short summary
=================
Returns the interface :ref:`ISimpleDateAndTimeAssertions`
with assert statements for date and time types with 32 bit length

.. <legal notes>

legal notes
=================
| SPDX-FileCopyrightText: © 2022 ekvip automation GmbH <info@ekvip.de>
| SPDX-License-Identifier: Apache-2.0
| For details check: Apache-2.0_

.. _Apache-2.0: https://www.apache.org/licenses/LICENSE-2.0

.. </legal notes>

methods
==================

*)

PROPERTY simple :ISimpleDateAndTimeAssertions
GET
simple := THIS^.assertionsFor32BitTypes;
END_GET
END_PROPERTY

END_FUNCTION_BLOCK

// ---- Assertor/Assertions/DateAndTimeAssertions/32Bit/classes/SimpleDateAndTimeAssertions.TcPOU
(*

short summary
=================
| This class provides assert statements for date and time types with 32 bit length
| It implements the interface :ref:`ISimpleDateAndTimeAssertions`
| For date and time (``DT``) use :ref:`SimpleDateAndTimeAssertions.dateAndTime`
| For date (``DATE``) use  :ref:`SimpleDateAndTimeAssertions.dateOnly`
| For time of day (``TOD``) use  :ref:`SimpleDateAndTimeAssertions.timeOfDay`

.. <legal notes>

legal notes
=================
| SPDX-FileCopyrightText: © 2022 ekvip automation GmbH <info@ekvip.de>
| SPDX-License-Identifier: Apache-2.0
| For details check: Apache-2.0_

.. _Apache-2.0: https://www.apache.org/licenses/LICENSE-2.0

.. </legal notes>

methods and properties
=======================

*)

{attribute 'reflection'}
FUNCTION_BLOCK INTERNAL SimpleDateAndTimeAssertions 
EXTENDS CNM_AbstractObject.Object
IMPLEMENTS ISimpleDateAndTimeAssertions, IAssertCallBacksetter
VAR
	(* class to handle date assertions *)
	dateAssertions		:DateAssertions32Bit();
	(* class to handle date and time assertions *)
	dateTimeAssertions	:DateTimeAssertions32Bit();
	(* class to handle time of day assertions *)
	timeOfDayAssertions	:TimeOfDayAssertions32Bit();
END_VAR

(*

short summary
=================
This abstract property returns the class name of the concrete object, 
It's for debugging purpose

.. <legal notes>

legal notes
=================
| SPDX-FileCopyrightText: © 2022 ekvip automation GmbH <info@ekvip.de>
| SPDX-License-Identifier: Apache-2.0
| For details check: Apache-2.0_

.. _Apache-2.0: https://www.apache.org/licenses/LICENSE-2.0

.. </legal notes>

*)

PROPERTY className :CNM_AbstractObject.ClassName
GET
className := 'CNM_AssertionInterfaceLib.SimplyDateAndTimeAssertions';
END_GET
END_PROPERTY

(*

short summary
=================
Returns the interface :ref:`I32BitDtAssertions`
with assert statements for 32 bit date and time ``DT``

.. <legal notes>

legal notes
=================
| SPDX-FileCopyrightText: © 2022 ekvip automation GmbH <info@ekvip.de>
| SPDX-License-Identifier: Apache-2.0
| For details check: Apache-2.0_

.. _Apache-2.0: https://www.apache.org/licenses/LICENSE-2.0

.. </legal notes>

*)

PROPERTY dateAndTime :I32BitDtAssertions
GET
dateAndTime := THIS^.dateTimeAssertions;
END_GET
END_PROPERTY

(*

short summary
=================
Returns the interface :ref:`I32BitDateAssertions`
with assert statements for 32 bit date ``DATE``

.. <legal notes>

legal notes
=================
| SPDX-FileCopyrightText: © 2022 ekvip automation GmbH <info@ekvip.de>
| SPDX-License-Identifier: Apache-2.0
| For details check: Apache-2.0_

.. _Apache-2.0: https://www.apache.org/licenses/LICENSE-2.0

.. </legal notes>

*)

PROPERTY dateOnly : I32BitDateAssertions
GET
dateOnly := THIS^.dateAssertions;
END_GET
END_PROPERTY

(*

short summary
=================
This methods is the setter for the callback class if an assertion was false

.. <legal notes>

legal notes
=================
| SPDX-FileCopyrightText: © 2022 ekvip automation GmbH <info@ekvip.de>
| SPDX-License-Identifier: Apache-2.0
| For details check: Apache-2.0_

.. _Apache-2.0: https://www.apache.org/licenses/LICENSE-2.0

.. </legal notes>

parameters
=================

*)

METHOD setCallBack
VAR_INPUT
	(* the class that must be informed if an assertion is false *)
	callBack	:IAssertCallback;  
END_VAR
THIS^.dateAssertions.setCallBack(callBack);
THIS^.dateTimeAssertions.setCallBack(callBack);
THIS^.timeOfDayAssertions.setCallBack(callBack);
END_METHOD

(*

short summary
=================
Returns the interface :ref:`I32BitDateAssertions`
with assert statements for 32 bit time of day ``TOD``

.. <legal notes>

legal notes
=================
| SPDX-FileCopyrightText: © 2022 ekvip automation GmbH <info@ekvip.de>
| SPDX-License-Identifier: Apache-2.0
| For details check: Apache-2.0_

.. _Apache-2.0: https://www.apache.org/licenses/LICENSE-2.0

.. </legal notes>

*)

PROPERTY timeOfDay :I32BitTodAssertions
GET
timeOfDay := THIS^.timeOfDayAssertions;
END_GET
END_PROPERTY

END_FUNCTION_BLOCK

// ---- Assertor/Assertions/DateAndTimeAssertions/32Bit/Date/classes/DateAssertions32Bit.TcPOU
(*

short summary
=================
This class provides assert statements for 32 bit ``DATE``.
It implements :ref:`I32BitDateAssertions`

.. <legal notes>

legal notes
=================
| SPDX-FileCopyrightText: © 2022 ekvip automation GmbH <info@ekvip.de>
| SPDX-License-Identifier: Apache-2.0
| For details check: Apache-2.0_

.. _Apache-2.0: https://www.apache.org/licenses/LICENSE-2.0

.. </legal notes>

methods and properties
=======================

*)

{attribute 'reflection'}
FUNCTION_BLOCK INTERNAL DateAssertions32Bit EXTENDS AbstactAssertion IMPLEMENTS I32BitDateAssertions
VAR
END_VAR

(*

short summary
=================
This abstract property returns the class name of the concrete object, 
It's for debugging purpose

.. <legal notes>

legal notes
=================
| SPDX-FileCopyrightText: © 2022 ekvip automation GmbH <info@ekvip.de>
| SPDX-License-Identifier: Apache-2.0
| For details check: Apache-2.0_

.. _Apache-2.0: https://www.apache.org/licenses/LICENSE-2.0

.. </legal notes>

*)

PROPERTY className :CNM_AbstractObject.ClassName
GET
className := 'CNM_AssertionInterfaceLib.DateAssertions32Bit';
END_GET
END_PROPERTY

(*

short summary
=================
This assertion method checks if the current value is equal to the expected value

.. <legal notes>

legal notes
=================
| SPDX-FileCopyrightText: © 2022 ekvip automation GmbH <info@ekvip.de>
| SPDX-License-Identifier: Apache-2.0
| For details check: Apache-2.0_

.. _Apache-2.0: https://www.apache.org/licenses/LICENSE-2.0

.. </legal notes>

parameters
=================

*)

METHOD valueIsEqualTo
VAR_INPUT
	(* current value to check *)
	currentValue	:DATE;
	(* expected value to compare *)
	expectedValue	:DATE;
	(* message if the assertion is false *)
	message			:AssertMessage;
END_VAR
IF (currentValue <> expectedValue) THEN
	THIS^.assertionWasWrong(message, THIS^.getDebugInfo('valueIsEqualTo'));
END_IF
END_METHOD

(*

short summary
=================
This assertion method checks if the current value is greater than the less value

.. <legal notes>

legal notes
=================
| SPDX-FileCopyrightText: © 2022 ekvip automation GmbH <info@ekvip.de>
| SPDX-License-Identifier: Apache-2.0
| For details check: Apache-2.0_

.. _Apache-2.0: https://www.apache.org/licenses/LICENSE-2.0

.. </legal notes>

parameters
=================

*)

METHOD valueIsGreaterThan
VAR_INPUT
	(* current value to check *)
	currentValue	:DATE;
	(* less than lower limit *)
	lessValue		:DATE;
	(* message if the assertion is false *)
	message			:AssertMessage;
END_VAR
IF (currentValue <= lessValue) THEN
	THIS^.assertionWasWrong(message, THIS^.getDebugInfo('valueIsGreaterThan'));
END_IF
END_METHOD

(*

short summary
=================
This assertion method checks if the current value is inside a limit

.. attention:: 
	limits are included: ``valueIsInRangeOf(date#1970-01-01, date#1970-01-01, date#1970-01-01)``
	is a true assertion

.. <legal notes>

legal notes
=================
| SPDX-FileCopyrightText: © 2022 ekvip automation GmbH <info@ekvip.de>
| SPDX-License-Identifier: Apache-2.0
| For details check: Apache-2.0_

.. _Apache-2.0: https://www.apache.org/licenses/LICENSE-2.0

.. </legal notes>

parameters
=================

*)

METHOD valueIsInRangeOf
VAR_INPUT
	(* lower limit for the current value *)
	lowerLimit		:DATE;
	(* current value to check *)
	currentValue	:DATE;
	(* upper limit for the current value *)
	upperLimit		:DATE;
	(* message if the assertion is false *)
	message			:AssertMessage;
END_VAR
IF (
	(currentValue < lowerLimit)
	OR (currentValue > upperLimit)
) THEN
	THIS^.assertionWasWrong(message, THIS^.getDebugInfo('valueIsInRangeOf'));
END_IF
END_METHOD

(*

short summary
=================
This assertion method checks if the current value is less than the greater value

.. <legal notes>

legal notes
=================
| SPDX-FileCopyrightText: © 2022 ekvip automation GmbH <info@ekvip.de>
| SPDX-License-Identifier: Apache-2.0
| For details check: Apache-2.0_

.. _Apache-2.0: https://www.apache.org/licenses/LICENSE-2.0

.. </legal notes>

parameters
=================

*)

METHOD valueIsLessThan
VAR_INPUT
	(* current value to check *)
	currentValue	:DATE;
	(* greater than upper limit *)
	greaterValue	:DATE;
	(* message if the assertion is false *)
	message			:AssertMessage;
END_VAR
IF (currentValue >= greaterValue) THEN
	THIS^.assertionWasWrong(message, THIS^.getDebugInfo('valueIsLessThan'));
END_IF
END_METHOD

(*

short summary
=================
This assertion method checks if the current value is less than or equal to the maximum value

.. <legal notes>

legal notes
=================
| SPDX-FileCopyrightText: © 2022 ekvip automation GmbH <info@ekvip.de>
| SPDX-License-Identifier: Apache-2.0
| For details check: Apache-2.0_

.. _Apache-2.0: https://www.apache.org/licenses/LICENSE-2.0

.. </legal notes>

parameters
=================

*)

METHOD valueIsMax
VAR_INPUT
	(* current value to check *)
	currentValue	:DATE;
	(* upper limit for the current value *)
	maximumValue	:DATE;
	(* message if the assertion is false *)
	message			:AssertMessage;
END_VAR
IF (currentValue > maximumValue) THEN
	THIS^.assertionWasWrong(message, THIS^.getDebugInfo('valueIsMax'));
END_IF
END_METHOD

(*

short summary
=================
This assertion method checks if the current value is greater than or equal to the minimum value

.. <legal notes>

legal notes
=================
| SPDX-FileCopyrightText: © 2022 ekvip automation GmbH <info@ekvip.de>
| SPDX-License-Identifier: Apache-2.0
| For details check: Apache-2.0_

.. _Apache-2.0: https://www.apache.org/licenses/LICENSE-2.0

.. </legal notes>

parameters
=================

*)

METHOD valueIsMin
VAR_INPUT
	(* current value to check *)
	currentValue	:DATE;
	(* lower limit for the current value *)
	minimumValue	:DATE;
	(* message if the assertion is false *)
	message			:AssertMessage;
END_VAR
IF (currentValue < minimumValue) THEN
	THIS^.assertionWasWrong(message, THIS^.getDebugInfo('valueIsMin'));
END_IF
END_METHOD

(*

short summary
=================
This assertion method checks if the current value is not equal to the unexpected value

.. <legal notes>

legal notes
=================
| SPDX-FileCopyrightText: © 2022 ekvip automation GmbH <info@ekvip.de>
| SPDX-License-Identifier: Apache-2.0
| For details check: Apache-2.0_

.. _Apache-2.0: https://www.apache.org/licenses/LICENSE-2.0

.. </legal notes>

parameters
=================

*)

METHOD valueIsNotEqualTo
VAR_INPUT
	(* current value to check *)
	currentValue	:DATE;
	(* unexpected value to compare *)
	unexpectedValue	:DATE;
	(* message if the assertion is false *)
	message			:AssertMessage;
END_VAR
IF (currentValue = unexpectedValue) THEN
	THIS^.assertionWasWrong(message, THIS^.getDebugInfo('valueIsNotEqualTo'));
END_IF
END_METHOD

END_FUNCTION_BLOCK

// ---- Assertor/Assertions/DateAndTimeAssertions/32Bit/DT/classes/DateTimeAssertions32Bit.TcPOU
(*

short summary
=================
This class provides assert statements for 32 bit date and time ``DT``.
It implements the interface :ref:`I32BitDtAssertions` 

.. <legal notes>

legal notes
=================
| SPDX-FileCopyrightText: © 2022 ekvip automation GmbH <info@ekvip.de>
| SPDX-License-Identifier: Apache-2.0
| For details check: Apache-2.0_

.. _Apache-2.0: https://www.apache.org/licenses/LICENSE-2.0

.. </legal notes>

methods and properties
=======================

*)

{attribute 'reflection'}
FUNCTION_BLOCK INTERNAL DateTimeAssertions32Bit EXTENDS AbstactAssertion IMPLEMENTS I32BitDtAssertions
VAR
END_VAR

(*

short summary
=================
This abstract property returns the class name of the concrete object, 
It's for debugging purpose

.. <legal notes>

legal notes
=================
| SPDX-FileCopyrightText: © 2022 ekvip automation GmbH <info@ekvip.de>
| SPDX-License-Identifier: Apache-2.0
| For details check: Apache-2.0_

.. _Apache-2.0: https://www.apache.org/licenses/LICENSE-2.0

.. </legal notes>

*)

PROPERTY className :CNM_AbstractObject.ClassName
GET
className := 'CNM_AssertionInterfaceLib.DateTimeAssertions32Bit';
END_GET
END_PROPERTY

(*

short summary
=================
This assertion method checks if the current value is equal to the expected value

.. <legal notes>

legal notes
=================
| SPDX-FileCopyrightText: © 2022 ekvip automation GmbH <info@ekvip.de>
| SPDX-License-Identifier: Apache-2.0
| For details check: Apache-2.0_

.. _Apache-2.0: https://www.apache.org/licenses/LICENSE-2.0

.. </legal notes>

parameters
=================

*)

METHOD valueIsEqualTo
VAR_INPUT
	(* current value to check *)
	currentValue	:DT;
	(* expected value to compare *)
	expectedValue	:DT;
	(* message if the assertion is false *)
	message			:AssertMessage;
END_VAR
IF (currentValue <> expectedValue) THEN
	THIS^.assertionWasWrong(message, THIS^.getDebugInfo('valueIsEqualTo'));
END_IF
END_METHOD

(*

short summary
=================
This assertion method checks if the current value is greater than the less value

.. <legal notes>

legal notes
=================
| SPDX-FileCopyrightText: © 2022 ekvip automation GmbH <info@ekvip.de>
| SPDX-License-Identifier: Apache-2.0
| For details check: Apache-2.0_

.. _Apache-2.0: https://www.apache.org/licenses/LICENSE-2.0

.. </legal notes>

parameters
=================

*)

METHOD valueIsGreaterThan
VAR_INPUT
	(* current value to check *)
	currentValue	:DT;
	(* less than lower limit *)
	lessValue		:DT;
	(* message if the assertion is false *)
	message			:AssertMessage;
END_VAR
IF (currentValue <= lessValue) THEN
	THIS^.assertionWasWrong(message, THIS^.getDebugInfo('valueIsGreaterThan'));
END_IF
END_METHOD

(*

short summary
=================
This assertion method checks if the current value is inside a limit

.. attention:: 
	limits are included: ``valueIsInRangeOf(dt#1970-01-01-0:0:0, dt#1970-01-01-0:0:0, dt#1970-01-01-0:0:0)``
	is a true assertion

.. <legal notes>

legal notes
=================
| SPDX-FileCopyrightText: © 2022 ekvip automation GmbH <info@ekvip.de>
| SPDX-License-Identifier: Apache-2.0
| For details check: Apache-2.0_

.. _Apache-2.0: https://www.apache.org/licenses/LICENSE-2.0

.. </legal notes>

parameters
=================

*)

METHOD valueIsInRangeOf
VAR_INPUT
	(* lower limit for the current value *)
	lowerLimit		:DT;
	(* current value to check *)
	currentValue	:DT;
	(* upper limit for the current value *)
	upperLimit		:DT;
	(* message if the assertion is false *)
	message			:AssertMessage;
END_VAR
IF (
	(currentValue < lowerLimit)
	OR (currentValue > upperLimit)
) THEN
	THIS^.assertionWasWrong(message, THIS^.getDebugInfo('valueIsInRangeOf'));
END_IF
END_METHOD

(*

short summary
=================
This assertion method checks if the current value is less than the greater value

.. <legal notes>

legal notes
=================
| SPDX-FileCopyrightText: © 2022 ekvip automation GmbH <info@ekvip.de>
| SPDX-License-Identifier: Apache-2.0
| For details check: Apache-2.0_

.. _Apache-2.0: https://www.apache.org/licenses/LICENSE-2.0

.. </legal notes>

parameters
=================

*)

METHOD valueIsLessThan
VAR_INPUT
	(* current value to check *)
	currentValue	:DT;
	(* greater than upper limit *)
	greaterValue	:DT;
	(* message if the assertion is false *)
	message			:AssertMessage;
END_VAR
IF (currentValue >= greaterValue) THEN
	THIS^.assertionWasWrong(message, THIS^.getDebugInfo('valueIsLessThan'));
END_IF
END_METHOD

(*

short summary
=================
This assertion method checks if the current value is less than or equal to the maximum value

.. <legal notes>

legal notes
=================
| SPDX-FileCopyrightText: © 2022 ekvip automation GmbH <info@ekvip.de>
| SPDX-License-Identifier: Apache-2.0
| For details check: Apache-2.0_

.. _Apache-2.0: https://www.apache.org/licenses/LICENSE-2.0

.. </legal notes>

parameters
=================

*)

METHOD valueIsMax
VAR_INPUT
	(* current value to check *)
	currentValue	:DT;
	(* upper limit for the current value *)
	maximumValue	:DT;
	(* message if the assertion is false *)
	message			:AssertMessage;
END_VAR
IF (currentValue > maximumValue) THEN
	THIS^.assertionWasWrong(message, THIS^.getDebugInfo('valueIsMax'));
END_IF
END_METHOD

(*

short summary
=================
This assertion method checks if the current value is greater than or equal to the minimum value

.. <legal notes>

legal notes
=================
| SPDX-FileCopyrightText: © 2022 ekvip automation GmbH <info@ekvip.de>
| SPDX-License-Identifier: Apache-2.0
| For details check: Apache-2.0_

.. _Apache-2.0: https://www.apache.org/licenses/LICENSE-2.0

.. </legal notes>

parameters
=================

*)

METHOD valueIsMin
VAR_INPUT
	(* current value to check *)
	currentValue	:DT;
	(* lower limit for the current value *)
	minimumValue	:DT;
	(* message if the assertion is false *)
	message			:AssertMessage;
END_VAR
IF (currentValue < minimumValue) THEN
	THIS^.assertionWasWrong(message, THIS^.getDebugInfo('valueIsMin'));
END_IF
END_METHOD

(*

short summary
=================
This assertion method checks if the current value is not equal to the unexpected value

.. <legal notes>

legal notes
=================
| SPDX-FileCopyrightText: © 2022 ekvip automation GmbH <info@ekvip.de>
| SPDX-License-Identifier: Apache-2.0
| For details check: Apache-2.0_

.. _Apache-2.0: https://www.apache.org/licenses/LICENSE-2.0

.. </legal notes>

parameters
=================

*)

METHOD valueIsNotEqualTo
VAR_INPUT
	(* current value to check *)
	currentValue	:DT;
	(* unexpected value to compare *)
	unexpectedValue	:DT;
	(* message if the assertion is false *)
	message			:AssertMessage;
END_VAR
IF (currentValue = unexpectedValue) THEN
	THIS^.assertionWasWrong(message, THIS^.getDebugInfo('valueIsNotEqualTo'));
END_IF
END_METHOD

END_FUNCTION_BLOCK

// ---- Assertor/Assertions/DateAndTimeAssertions/32Bit/TOD/classes/TimeOfDayAssertions32Bit.TcPOU
(*

short summary
=================
This class provides assert statements for 32 bit time of day ``TOD``.
It implements the interface :ref:`I32BitTodAssertions`

.. <legal notes>

legal notes
=================
| SPDX-FileCopyrightText: © 2022 ekvip automation GmbH <info@ekvip.de>
| SPDX-License-Identifier: Apache-2.0
| For details check: Apache-2.0_

.. _Apache-2.0: https://www.apache.org/licenses/LICENSE-2.0

.. </legal notes>

methods
==================

*)

{attribute 'reflection'}
FUNCTION_BLOCK INTERNAL TimeOfDayAssertions32Bit EXTENDS AbstactAssertion IMPLEMENTS I32BitTodAssertions
VAR
END_VAR

(*

short summary
=================
This abstract property returns the class name of the concrete object, 
It's for debugging purpose

.. <legal notes>

legal notes
=================
| SPDX-FileCopyrightText: © 2022 ekvip automation GmbH <info@ekvip.de>
| SPDX-License-Identifier: Apache-2.0
| For details check: Apache-2.0_

.. _Apache-2.0: https://www.apache.org/licenses/LICENSE-2.0

.. </legal notes>

*)

PROPERTY className :CNM_AbstractObject.ClassName
GET
className := 'CNM_AssertionInterfaceLib.TimeOfDayAssertions32Bit';
END_GET
END_PROPERTY

(*

short summary
=================
This assertion method checks if the current value is equal to the expected value

.. <legal notes>

legal notes
=================
| SPDX-FileCopyrightText: © 2022 ekvip automation GmbH <info@ekvip.de>
| SPDX-License-Identifier: Apache-2.0
| For details check: Apache-2.0_

.. _Apache-2.0: https://www.apache.org/licenses/LICENSE-2.0

.. </legal notes>

parameters
=================

*)

METHOD valueIsEqualTo
VAR_INPUT
	(* current value to check *)
	currentValue	:TOD;
	(* expected value to compare *)
	expectedValue	:TOD;
	(* message if the assertion is false *)
	message			:AssertMessage;
END_VAR
IF (currentValue <> expectedValue) THEN
	THIS^.assertionWasWrong(message, THIS^.getDebugInfo('valueIsEqualTo'));
END_IF
END_METHOD

(*

short summary
=================
This assertion method checks if the current value is greater than the less value

.. <legal notes>

legal notes
=================
| SPDX-FileCopyrightText: © 2022 ekvip automation GmbH <info@ekvip.de>
| SPDX-License-Identifier: Apache-2.0
| For details check: Apache-2.0_

.. _Apache-2.0: https://www.apache.org/licenses/LICENSE-2.0

.. </legal notes>

parameters
=================

*)

METHOD valueIsGreaterThan
VAR_INPUT
	(* current value to check *)
	currentValue	:TOD;
	(* less than lower limit *)
	lessValue		:TOD;
	(* message if the assertion is false *)
	message			:AssertMessage;
END_VAR
IF (currentValue <= lessValue) THEN
	THIS^.assertionWasWrong(message, THIS^.getDebugInfo('valueIsGreaterThan'));
END_IF
END_METHOD

(*

short summary
=================
This assertion method checks if the current value is inside a limit

.. attention:: 
	limits are included: ``valueIsInRangeOf(tod#3:0:0, tod#3:0:0, tod#3:0:0)`` is a true assertion

.. <legal notes>

legal notes
=================
| SPDX-FileCopyrightText: © 2022 ekvip automation GmbH <info@ekvip.de>
| SPDX-License-Identifier: Apache-2.0
| For details check: Apache-2.0_

.. _Apache-2.0: https://www.apache.org/licenses/LICENSE-2.0

.. </legal notes>

parameters
=================

*)

METHOD valueIsInRangeOf
VAR_INPUT
	(* lower limit for the current value *)
	lowerLimit		:TOD;
	(* current value to check *)
	currentValue	:TOD;
	(* upper limit for the current value *)
	upperLimit		:TOD;
	(* message if the assertion is false *)
	message			:AssertMessage;
END_VAR
IF (
	(currentValue < lowerLimit)
	OR (currentValue > upperLimit)
) THEN
	THIS^.assertionWasWrong(message, THIS^.getDebugInfo('valueIsInRangeOf'));
END_IF
END_METHOD

(*

short summary
=================
This assertion method checks if the current value is less than the greater value

.. <legal notes>

legal notes
=================
| SPDX-FileCopyrightText: © 2022 ekvip automation GmbH <info@ekvip.de>
| SPDX-License-Identifier: Apache-2.0
| For details check: Apache-2.0_

.. _Apache-2.0: https://www.apache.org/licenses/LICENSE-2.0

.. </legal notes>

parameters
=================

*)

METHOD valueIsLessThan
VAR_INPUT
	(* current value to check *)
	currentValue	:TOD;
	(* greater than upper limit *)
	greaterValue	:TOD;
	(* message if the assertion is false *)
	message			:AssertMessage;
END_VAR
IF (currentValue >= greaterValue) THEN
	THIS^.assertionWasWrong(message, THIS^.getDebugInfo('valueIsLessThan'));
END_IF
END_METHOD

(*

short summary
=================
This assertion method checks if the current value is less than or equal to the maximum value

.. <legal notes>

legal notes
=================
| SPDX-FileCopyrightText: © 2022 ekvip automation GmbH <info@ekvip.de>
| SPDX-License-Identifier: Apache-2.0
| For details check: Apache-2.0_

.. _Apache-2.0: https://www.apache.org/licenses/LICENSE-2.0

.. </legal notes>

parameters
=================

*)

METHOD valueIsMax
VAR_INPUT
	(* current value to check *)
	currentValue	:TOD;
	(* upper limit for the current value *)
	maximumValue	:TOD;
	(* message if the assertion is false *)
	message			:AssertMessage;
END_VAR
IF (currentValue > maximumValue) THEN
	THIS^.assertionWasWrong(message, THIS^.getDebugInfo('valueIsMax'));
END_IF
END_METHOD

(*

short summary
=================
This assertion method checks if the current value is greater than or equal to the minimum value

.. <legal notes>

legal notes
=================
| SPDX-FileCopyrightText: © 2022 ekvip automation GmbH <info@ekvip.de>
| SPDX-License-Identifier: Apache-2.0
| For details check: Apache-2.0_

.. _Apache-2.0: https://www.apache.org/licenses/LICENSE-2.0

.. </legal notes>

parameters
=================

*)

METHOD valueIsMin
VAR_INPUT
	(* current value to check *)
	currentValue	:TOD;
	(* lower limit for the current value *)
	minimumValue	:TOD;
	(* message if the assertion is false *)
	message			:AssertMessage;
END_VAR
IF (currentValue < minimumValue) THEN
	THIS^.assertionWasWrong(message, THIS^.getDebugInfo('valueIsMin'));
END_IF
END_METHOD

(*

short summary
=================
This assertion method checks if the current value is not equal to the unexpected value

.. <legal notes>

legal notes
=================
| SPDX-FileCopyrightText: © 2022 ekvip automation GmbH <info@ekvip.de>
| SPDX-License-Identifier: Apache-2.0
| For details check: Apache-2.0_

.. _Apache-2.0: https://www.apache.org/licenses/LICENSE-2.0

.. </legal notes>

parameters
=================

*)

METHOD valueIsNotEqualTo
VAR_INPUT
	(* current value to check *)
	currentValue	:TOD;
	(* unexpected value to compare *)
	unexpectedValue	:TOD;
	(* message if the assertion is false *)
	message			:AssertMessage;
END_VAR
IF (currentValue = unexpectedValue) THEN
	THIS^.assertionWasWrong(message, THIS^.getDebugInfo('valueIsNotEqualTo'));
END_IF
END_METHOD

END_FUNCTION_BLOCK

// ---- Assertor/Assertions/DateAndTimeAssertions/64Bit/classes/LongDateAndTimeAssertions.TcPOU
(*

short summary
=================
| This class provides assert statements for date and time types with 32 bit length
| It implements the interface :ref:`ISimpleDateAndTimeAssertions`
| For date and time (``DT``) use :ref:`SimpleDateAndTimeAssertions.dateAndTime`
| For date (``DATE``) use  :ref:`SimpleDateAndTimeAssertions.dateOnly`
| For time of day (``TOD``) use  :ref:`SimpleDateAndTimeAssertions.timeOfDay`

.. <legal notes>

legal notes
=================
| SPDX-FileCopyrightText: © 2022 ekvip automation GmbH <info@ekvip.de>
| SPDX-License-Identifier: Apache-2.0
| For details check: Apache-2.0_

.. _Apache-2.0: https://www.apache.org/licenses/LICENSE-2.0

.. </legal notes>

methods and properties
=======================

*)

{attribute 'reflection'}
FUNCTION_BLOCK INTERNAL LongDateAndTimeAssertions 
EXTENDS CNM_AbstractObject.Object
IMPLEMENTS ILongDateAndTimeAssertions, IAssertCallBacksetter
VAR
	(* class to handle date assertions *)
	dateAssertions		:DateAssertions64Bit();
	(* class to handle date and time assertions *)
	dateTimeAssertions	:DateTimeAssertions64Bit();
	(* class to handle time of day assertions *)
	timeOfDayAssertions	:TimeOfDayAssertions64Bit();
END_VAR

(*

short summary
=================
This abstract property returns the class name of the concrete object, 
It's for debugging purpose

.. <legal notes>

legal notes
=================
| SPDX-FileCopyrightText: © 2022 ekvip automation GmbH <info@ekvip.de>
| SPDX-License-Identifier: Apache-2.0
| For details check: Apache-2.0_

.. _Apache-2.0: https://www.apache.org/licenses/LICENSE-2.0

.. </legal notes>

*)

PROPERTY className :CNM_AbstractObject.ClassName
GET
className := 'CNM_AssertionInterfaceLib.SimplyDateAndTimeAssertions';
END_GET
END_PROPERTY

(*

short summary
=================
Returns the interface :ref:`I32BitDtAssertions`
with assert statements for 32 bit date and time ``DT``

.. <legal notes>

legal notes
=================
| SPDX-FileCopyrightText: © 2022 ekvip automation GmbH <info@ekvip.de>
| SPDX-License-Identifier: Apache-2.0
| For details check: Apache-2.0_

.. _Apache-2.0: https://www.apache.org/licenses/LICENSE-2.0

.. </legal notes>

*)

PROPERTY dateAndTime :I64BitDtAssertions
GET
dateAndTime := THIS^.dateTimeAssertions;
END_GET
END_PROPERTY

(*

short summary
=================
Returns the interface :ref:`I32BitDateAssertions`
with assert statements for 32 bit date ``DATE``

.. <legal notes>

legal notes
=================
| SPDX-FileCopyrightText: © 2022 ekvip automation GmbH <info@ekvip.de>
| SPDX-License-Identifier: Apache-2.0
| For details check: Apache-2.0_

.. _Apache-2.0: https://www.apache.org/licenses/LICENSE-2.0

.. </legal notes>

*)

PROPERTY dateOnly : I64BitDateAssertions
GET
dateOnly := THIS^.dateAssertions;
END_GET
END_PROPERTY

(*

short summary
=================
This methods is the setter for the callback class if an assertion was false

.. <legal notes>

legal notes
=================
| SPDX-FileCopyrightText: © 2022 ekvip automation GmbH <info@ekvip.de>
| SPDX-License-Identifier: Apache-2.0
| For details check: Apache-2.0_

.. _Apache-2.0: https://www.apache.org/licenses/LICENSE-2.0

.. </legal notes>

parameters
=================

*)

METHOD setCallBack
VAR_INPUT
	(* the class that must be informed if an assertion is false *)
	callBack	:IAssertCallback;  
END_VAR
THIS^.dateAssertions.setCallBack(callBack);
THIS^.dateTimeAssertions.setCallBack(callBack);
THIS^.timeOfDayAssertions.setCallBack(callBack);
END_METHOD

(*

short summary
=================
Returns the interface :ref:`I32BitDateAssertions`
with assert statements for 32 bit time of day ``TOD``

.. <legal notes>

legal notes
=================
| SPDX-FileCopyrightText: © 2022 ekvip automation GmbH <info@ekvip.de>
| SPDX-License-Identifier: Apache-2.0
| For details check: Apache-2.0_

.. _Apache-2.0: https://www.apache.org/licenses/LICENSE-2.0

.. </legal notes>

*)

PROPERTY timeOfDay :I64BitTodAssertions
GET
timeOfDay := THIS^.timeOfDayAssertions;
END_GET
END_PROPERTY

END_FUNCTION_BLOCK

// ---- Assertor/Assertions/DateAndTimeAssertions/64Bit/LDate/classes/DateAssertions64Bit.TcPOU
(*

short summary
=================
This class provides assert statements for 64 bit ``LDATE``.
It implements :ref:`I64BitDateAssertions`

.. <legal notes>

legal notes
=================
| SPDX-FileCopyrightText: © 2022 ekvip automation GmbH <info@ekvip.de>
| SPDX-License-Identifier: Apache-2.0
| For details check: Apache-2.0_

.. _Apache-2.0: https://www.apache.org/licenses/LICENSE-2.0

.. </legal notes>

methods and properties
=======================

*)

{attribute 'reflection'}
FUNCTION_BLOCK INTERNAL DateAssertions64Bit EXTENDS AbstactAssertion IMPLEMENTS I64BitDateAssertions
VAR
END_VAR

(*

short summary
=================
This abstract property returns the class name of the concrete object, 
It's for debugging purpose

.. <legal notes>

legal notes
=================
| SPDX-FileCopyrightText: © 2022 ekvip automation GmbH <info@ekvip.de>
| SPDX-License-Identifier: Apache-2.0
| For details check: Apache-2.0_

.. _Apache-2.0: https://www.apache.org/licenses/LICENSE-2.0

.. </legal notes>

*)

PROPERTY className :CNM_AbstractObject.ClassName
GET
className := 'CNM_AssertionInterfaceLib.DateAssertions32Bit';
END_GET
END_PROPERTY

(*

short summary
=================
This assertion method checks if the current value is equal to the expected value

.. <legal notes>

legal notes
=================
| SPDX-FileCopyrightText: © 2022 ekvip automation GmbH <info@ekvip.de>
| SPDX-License-Identifier: Apache-2.0
| For details check: Apache-2.0_

.. _Apache-2.0: https://www.apache.org/licenses/LICENSE-2.0

.. </legal notes>

parameters
=================

*)

METHOD valueIsEqualTo
VAR_INPUT
	(* current value to check *)
	currentValue	:LDATE;
	(* expected value to compare *)
	expectedValue	:LDATE;
	(* message if the assertion is false *)
	message			:AssertMessage;
END_VAR
IF (currentValue <> expectedValue) THEN
	THIS^.assertionWasWrong(message, THIS^.getDebugInfo('valueIsEqualTo'));
END_IF
END_METHOD

(*

short summary
=================
This assertion method checks if the current value is greater than the less value

.. <legal notes>

legal notes
=================
| SPDX-FileCopyrightText: © 2022 ekvip automation GmbH <info@ekvip.de>
| SPDX-License-Identifier: Apache-2.0
| For details check: Apache-2.0_

.. _Apache-2.0: https://www.apache.org/licenses/LICENSE-2.0

.. </legal notes>

parameters
=================

*)

METHOD valueIsGreaterThan
VAR_INPUT
	(* current value to check *)
	currentValue	:LDATE;
	(* less than lower limit *)
	lessValue		:LDATE;
	(* message if the assertion is false *)
	message			:AssertMessage;
END_VAR
IF (currentValue <= lessValue) THEN
	THIS^.assertionWasWrong(message, THIS^.getDebugInfo('valueIsGreaterThan'));
END_IF
END_METHOD

(*

short summary
=================
This assertion method checks if the current value is inside a limit

.. attention:: 
	limits are included: ``valueIsInRangeOf(ldate#1970-01-01, ldate#1970-01-01, ldate#1970-01-01)``
	is a true assertion

.. <legal notes>

legal notes
=================
| SPDX-FileCopyrightText: © 2022 ekvip automation GmbH <info@ekvip.de>
| SPDX-License-Identifier: Apache-2.0
| For details check: Apache-2.0_

.. _Apache-2.0: https://www.apache.org/licenses/LICENSE-2.0

.. </legal notes>

parameters
=================

*)

METHOD valueIsInRangeOf
VAR_INPUT
	(* lower limit for the current value *)
	lowerLimit		:LDATE;
	(* current value to check *)
	currentValue	:LDATE;
	(* upper limit for the current value *)
	upperLimit		:LDATE;
	(* message if the assertion is false *)
	message			:AssertMessage;
END_VAR
IF (
	(currentValue < lowerLimit)
	OR (currentValue > upperLimit)
) THEN
	THIS^.assertionWasWrong(message, THIS^.getDebugInfo('valueIsInRangeOf'));
END_IF
END_METHOD

(*

short summary
=================
This assertion method checks if the current value is less than the greater value

.. <legal notes>

legal notes
=================
| SPDX-FileCopyrightText: © 2022 ekvip automation GmbH <info@ekvip.de>
| SPDX-License-Identifier: Apache-2.0
| For details check: Apache-2.0_

.. _Apache-2.0: https://www.apache.org/licenses/LICENSE-2.0

.. </legal notes>

parameters
=================

*)

METHOD valueIsLessThan
VAR_INPUT
	(* current value to check *)
	currentValue	:LDATE;
	(* greater than upper limit *)
	greaterValue	:LDATE;
	(* message if the assertion is false *)
	message			:AssertMessage;
END_VAR
IF (currentValue >= greaterValue) THEN
	THIS^.assertionWasWrong(message, THIS^.getDebugInfo('valueIsLessThan'));
END_IF
END_METHOD

(*

short summary
=================
This assertion method checks if the current value is less than or equal to the maximum value

.. <legal notes>

legal notes
=================
| SPDX-FileCopyrightText: © 2022 ekvip automation GmbH <info@ekvip.de>
| SPDX-License-Identifier: Apache-2.0
| For details check: Apache-2.0_

.. _Apache-2.0: https://www.apache.org/licenses/LICENSE-2.0

.. </legal notes>

parameters
=================

*)

METHOD valueIsMax
VAR_INPUT
	(* current value to check *)
	currentValue	:LDATE;
	(* upper limit for the current value *)
	maximumValue	:LDATE;
	(* message if the assertion is false *)
	message			:AssertMessage;
END_VAR
IF (currentValue > maximumValue) THEN
	THIS^.assertionWasWrong(message, THIS^.getDebugInfo('valueIsMax'));
END_IF
END_METHOD

(*

short summary
=================
This assertion method checks if the current value is greater than or equal to the minimum value

.. <legal notes>

legal notes
=================
| SPDX-FileCopyrightText: © 2022 ekvip automation GmbH <info@ekvip.de>
| SPDX-License-Identifier: Apache-2.0
| For details check: Apache-2.0_

.. _Apache-2.0: https://www.apache.org/licenses/LICENSE-2.0

.. </legal notes>

parameters
=================

*)

METHOD valueIsMin
VAR_INPUT
	(* current value to check *)
	currentValue	:LDATE;
	(* lower limit for the current value *)
	minimumValue	:LDATE;
	(* message if the assertion is false *)
	message			:AssertMessage;
END_VAR
IF (currentValue < minimumValue) THEN
	THIS^.assertionWasWrong(message, THIS^.getDebugInfo('valueIsMin'));
END_IF
END_METHOD

(*

short summary
=================
This assertion method checks if the current value is not equal to the unexpected value

.. <legal notes>

legal notes
=================
| SPDX-FileCopyrightText: © 2022 ekvip automation GmbH <info@ekvip.de>
| SPDX-License-Identifier: Apache-2.0
| For details check: Apache-2.0_

.. _Apache-2.0: https://www.apache.org/licenses/LICENSE-2.0

.. </legal notes>

parameters
=================

*)

METHOD valueIsNotEqualTo
VAR_INPUT
	(* current value to check *)
	currentValue	:LDATE;
	(* unexpected value to compare *)
	unexpectedValue	:LDATE;
	(* message if the assertion is false *)
	message			:AssertMessage;
END_VAR
IF (currentValue = unexpectedValue) THEN
	THIS^.assertionWasWrong(message, THIS^.getDebugInfo('valueIsNotEqualTo'));
END_IF
END_METHOD

END_FUNCTION_BLOCK

// ---- Assertor/Assertions/DateAndTimeAssertions/64Bit/LDT/classes/DateTimeAssertions64Bit.TcPOU
(*

short summary
=================
This class provides assert statements for 64 bit date and time ``LDT``.
It implements the interface :ref:`I64BitDtAssertions` 

.. <legal notes>

legal notes
=================
| SPDX-FileCopyrightText: © 2022 ekvip automation GmbH <info@ekvip.de>
| SPDX-License-Identifier: Apache-2.0
| For details check: Apache-2.0_

.. _Apache-2.0: https://www.apache.org/licenses/LICENSE-2.0

.. </legal notes>

methods and properties
=======================

*)

{attribute 'reflection'}
FUNCTION_BLOCK INTERNAL DateTimeAssertions64Bit EXTENDS AbstactAssertion IMPLEMENTS I64BitDtAssertions
VAR
END_VAR

(*

short summary
=================
This abstract property returns the class name of the concrete object, 
It's for debugging purpose

.. <legal notes>

legal notes
=================
| SPDX-FileCopyrightText: © 2022 ekvip automation GmbH <info@ekvip.de>
| SPDX-License-Identifier: Apache-2.0
| For details check: Apache-2.0_

.. _Apache-2.0: https://www.apache.org/licenses/LICENSE-2.0

.. </legal notes>

*)

PROPERTY className :CNM_AbstractObject.ClassName
GET
className := 'CNM_AssertionInterfaceLib.DateTimeAssertions64Bit';
END_GET
END_PROPERTY

(*

short summary
=================
This assertion method checks if the current value is equal to the expected value

.. <legal notes>

legal notes
=================
| SPDX-FileCopyrightText: © 2022 ekvip automation GmbH <info@ekvip.de>
| SPDX-License-Identifier: Apache-2.0
| For details check: Apache-2.0_

.. _Apache-2.0: https://www.apache.org/licenses/LICENSE-2.0

.. </legal notes>

parameters
=================

*)

METHOD valueIsEqualTo
VAR_INPUT
	(* current value to check *)
	currentValue	:LDT;
	(* expected value to compare *)
	expectedValue	:LDT;
	(* message if the assertion is false *)
	message			:AssertMessage;
END_VAR
IF (currentValue <> expectedValue) THEN
	THIS^.assertionWasWrong(message, THIS^.getDebugInfo('valueIsEqualTo'));
END_IF
END_METHOD

(*

short summary
=================
This assertion method checks if the current value is greater than the less value

.. <legal notes>

legal notes
=================
| SPDX-FileCopyrightText: © 2022 ekvip automation GmbH <info@ekvip.de>
| SPDX-License-Identifier: Apache-2.0
| For details check: Apache-2.0_

.. _Apache-2.0: https://www.apache.org/licenses/LICENSE-2.0

.. </legal notes>

parameters
=================

*)

METHOD valueIsGreaterThan
VAR_INPUT
	(* current value to check *)
	currentValue	:LDT;
	(* less than lower limit *)
	lessValue		:LDT;
	(* message if the assertion is false *)
	message			:AssertMessage;
END_VAR
IF (currentValue <= lessValue) THEN
	THIS^.assertionWasWrong(message, THIS^.getDebugInfo('valueIsGreaterThan'));
END_IF
END_METHOD

(*

short summary
=================
This assertion method checks if the current value is inside a limit

.. attention:: 
	limits are included: ``valueIsInRangeOf(ldt#1970-01-01-0:0:0, ldt#1970-01-01-0:0:0, ldt#1970-01-01-0:0:0)``
	is a true assertion

.. <legal notes>

legal notes
=================
| SPDX-FileCopyrightText: © 2022 ekvip automation GmbH <info@ekvip.de>
| SPDX-License-Identifier: Apache-2.0
| For details check: Apache-2.0_

.. _Apache-2.0: https://www.apache.org/licenses/LICENSE-2.0

.. </legal notes>

parameters
=================

*)

METHOD valueIsInRangeOf
VAR_INPUT
	(* lower limit for the current value *)
	lowerLimit		:LDT;
	(* current value to check *)
	currentValue	:LDT;
	(* upper limit for the current value *)
	upperLimit		:LDT;
	(* message if the assertion is false *)
	message			:AssertMessage;
END_VAR
IF (
	(currentValue < lowerLimit)
	OR (currentValue > upperLimit)
) THEN
	THIS^.assertionWasWrong(message, THIS^.getDebugInfo('valueIsInRangeOf'));
END_IF
END_METHOD

(*

short summary
=================
This assertion method checks if the current value is less than the greater value

.. <legal notes>

legal notes
=================
| SPDX-FileCopyrightText: © 2022 ekvip automation GmbH <info@ekvip.de>
| SPDX-License-Identifier: Apache-2.0
| For details check: Apache-2.0_

.. _Apache-2.0: https://www.apache.org/licenses/LICENSE-2.0

.. </legal notes>

parameters
=================

*)

METHOD valueIsLessThan
VAR_INPUT
	(* current value to check *)
	currentValue	:LDT;
	(* greater than upper limit *)
	greaterValue	:LDT;
	(* message if the assertion is false *)
	message			:AssertMessage;
END_VAR
IF (currentValue >= greaterValue) THEN
	THIS^.assertionWasWrong(message, THIS^.getDebugInfo('valueIsLessThan'));
END_IF
END_METHOD

(*

short summary
=================
This assertion method checks if the current value is less than or equal to the maximum value

.. <legal notes>

legal notes
=================
| SPDX-FileCopyrightText: © 2022 ekvip automation GmbH <info@ekvip.de>
| SPDX-License-Identifier: Apache-2.0
| For details check: Apache-2.0_

.. _Apache-2.0: https://www.apache.org/licenses/LICENSE-2.0

.. </legal notes>

parameters
=================

*)

METHOD valueIsMax
VAR_INPUT
	(* current value to check *)
	currentValue	:LDT;
	(* upper limit for the current value *)
	maximumValue	:LDT;
	(* message if the assertion is false *)
	message			:AssertMessage;
END_VAR
IF (currentValue > maximumValue) THEN
	THIS^.assertionWasWrong(message, THIS^.getDebugInfo('valueIsMax'));
END_IF
END_METHOD

(*

short summary
=================
This assertion method checks if the current value is greater than or equal to the minimum value

.. <legal notes>

legal notes
=================
| SPDX-FileCopyrightText: © 2022 ekvip automation GmbH <info@ekvip.de>
| SPDX-License-Identifier: Apache-2.0
| For details check: Apache-2.0_

.. _Apache-2.0: https://www.apache.org/licenses/LICENSE-2.0

.. </legal notes>

parameters
=================

*)

METHOD valueIsMin
VAR_INPUT
	(* current value to check *)
	currentValue	:LDT;
	(* lower limit for the current value *)
	minimumValue	:LDT;
	(* message if the assertion is false *)
	message			:AssertMessage;
END_VAR
IF (currentValue < minimumValue) THEN
	THIS^.assertionWasWrong(message, THIS^.getDebugInfo('valueIsMin'));
END_IF
END_METHOD

(*

short summary
=================
This assertion method checks if the current value is not equal to the unexpected value

.. <legal notes>

legal notes
=================
| SPDX-FileCopyrightText: © 2022 ekvip automation GmbH <info@ekvip.de>
| SPDX-License-Identifier: Apache-2.0
| For details check: Apache-2.0_

.. _Apache-2.0: https://www.apache.org/licenses/LICENSE-2.0

.. </legal notes>

parameters
=================

*)

METHOD valueIsNotEqualTo
VAR_INPUT
	(* current value to check *)
	currentValue	:LDT;
	(* unexpected value to compare *)
	unexpectedValue	:LDT;
	(* message if the assertion is false *)
	message			:AssertMessage;
END_VAR
IF (currentValue = unexpectedValue) THEN
	THIS^.assertionWasWrong(message, THIS^.getDebugInfo('valueIsNotEqualTo'));
END_IF
END_METHOD

END_FUNCTION_BLOCK

// ---- Assertor/Assertions/DateAndTimeAssertions/64Bit/LTOD/classes/TimeOfDayAssertions64Bit.TcPOU
(*

short summary
=================
This class provides assert statements for 32 bit time of day ``LTOD``.
It implements the interface :ref:`I64BitTodAssertions`

.. <legal notes>

legal notes
=================
| SPDX-FileCopyrightText: © 2022 ekvip automation GmbH <info@ekvip.de>
| SPDX-License-Identifier: Apache-2.0
| For details check: Apache-2.0_

.. _Apache-2.0: https://www.apache.org/licenses/LICENSE-2.0

.. </legal notes>

methods
==================

*)

{attribute 'reflection'}
FUNCTION_BLOCK INTERNAL TimeOfDayAssertions64Bit EXTENDS AbstactAssertion IMPLEMENTS I64BitTodAssertions
VAR
END_VAR

(*

short summary
=================
This abstract property returns the class name of the concrete object, 
It's for debugging purpose

.. <legal notes>

legal notes
=================
| SPDX-FileCopyrightText: © 2022 ekvip automation GmbH <info@ekvip.de>
| SPDX-License-Identifier: Apache-2.0
| For details check: Apache-2.0_

.. _Apache-2.0: https://www.apache.org/licenses/LICENSE-2.0

.. </legal notes>

*)

PROPERTY className :CNM_AbstractObject.ClassName
GET
className := 'CNM_AssertionInterfaceLib.TimeOfDayAssertions64Bit';
END_GET
END_PROPERTY

(*

short summary
=================
This assertion method checks if the current value is equal to the expected value

.. <legal notes>

legal notes
=================
| SPDX-FileCopyrightText: © 2022 ekvip automation GmbH <info@ekvip.de>
| SPDX-License-Identifier: Apache-2.0
| For details check: Apache-2.0_

.. _Apache-2.0: https://www.apache.org/licenses/LICENSE-2.0

.. </legal notes>

parameters
=================

*)

METHOD valueIsEqualTo
VAR_INPUT
	(* current value to check *)
	currentValue	:LTOD;
	(* expected value to compare *)
	expectedValue	:LTOD;
	(* message if the assertion is false *)
	message			:AssertMessage;
END_VAR
IF (currentValue <> expectedValue) THEN
	THIS^.assertionWasWrong(message, THIS^.getDebugInfo('valueIsEqualTo'));
END_IF
END_METHOD

(*

short summary
=================
This assertion method checks if the current value is greater than the less value

.. <legal notes>

legal notes
=================
| SPDX-FileCopyrightText: © 2022 ekvip automation GmbH <info@ekvip.de>
| SPDX-License-Identifier: Apache-2.0
| For details check: Apache-2.0_

.. _Apache-2.0: https://www.apache.org/licenses/LICENSE-2.0

.. </legal notes>

parameters
=================

*)

METHOD valueIsGreaterThan
VAR_INPUT
	(* current value to check *)
	currentValue	:LTOD;
	(* less than lower limit *)
	lessValue		:LTOD;
	(* message if the assertion is false *)
	message			:AssertMessage;
END_VAR
IF (currentValue <= lessValue) THEN
	THIS^.assertionWasWrong(message, THIS^.getDebugInfo('valueIsGreaterThan'));
END_IF
END_METHOD

(*

short summary
=================
This assertion method checks if the current value is inside a limit

.. attention:: 
	limits are included: ``valueIsInRangeOf(ltod#3:0:0, ltod#3:0:0, ltod#3:0:0)`` is a true assertion

.. <legal notes>

legal notes
=================
| SPDX-FileCopyrightText: © 2022 ekvip automation GmbH <info@ekvip.de>
| SPDX-License-Identifier: Apache-2.0
| For details check: Apache-2.0_

.. _Apache-2.0: https://www.apache.org/licenses/LICENSE-2.0

.. </legal notes>

parameters
=================

*)

METHOD valueIsInRangeOf
VAR_INPUT
	(* lower limit for the current value *)
	lowerLimit		:LTOD;
	(* current value to check *)
	currentValue	:LTOD;
	(* upper limit for the current value *)
	upperLimit		:LTOD;
	(* message if the assertion is false *)
	message			:AssertMessage;
END_VAR
IF (
	(currentValue < lowerLimit)
	OR (currentValue > upperLimit)
) THEN
	THIS^.assertionWasWrong(message, THIS^.getDebugInfo('valueIsInRangeOf'));
END_IF
END_METHOD

(*

short summary
=================
This assertion method checks if the current value is less than the greater value

.. <legal notes>

legal notes
=================
| SPDX-FileCopyrightText: © 2022 ekvip automation GmbH <info@ekvip.de>
| SPDX-License-Identifier: Apache-2.0
| For details check: Apache-2.0_

.. _Apache-2.0: https://www.apache.org/licenses/LICENSE-2.0

.. </legal notes>

parameters
=================

*)

METHOD valueIsLessThan
VAR_INPUT
	(* current value to check *)
	currentValue	:LTOD;
	(* greater than upper limit *)
	greaterValue	:LTOD;
	(* message if the assertion is false *)
	message			:AssertMessage;
END_VAR
IF (currentValue >= greaterValue) THEN
	THIS^.assertionWasWrong(message, THIS^.getDebugInfo('valueIsLessThan'));
END_IF
END_METHOD

(*

short summary
=================
This assertion method checks if the current value is less than or equal to the maximum value

.. <legal notes>

legal notes
=================
| SPDX-FileCopyrightText: © 2022 ekvip automation GmbH <info@ekvip.de>
| SPDX-License-Identifier: Apache-2.0
| For details check: Apache-2.0_

.. _Apache-2.0: https://www.apache.org/licenses/LICENSE-2.0

.. </legal notes>

parameters
=================

*)

METHOD valueIsMax
VAR_INPUT
	(* current value to check *)
	currentValue	:LTOD;
	(* upper limit for the current value *)
	maximumValue	:LTOD;
	(* message if the assertion is false *)
	message			:AssertMessage;
END_VAR
IF (currentValue > maximumValue) THEN
	THIS^.assertionWasWrong(message, THIS^.getDebugInfo('valueIsMax'));
END_IF
END_METHOD

(*

short summary
=================
This assertion method checks if the current value is greater than or equal to the minimum value

.. <legal notes>

legal notes
=================
| SPDX-FileCopyrightText: © 2022 ekvip automation GmbH <info@ekvip.de>
| SPDX-License-Identifier: Apache-2.0
| For details check: Apache-2.0_

.. _Apache-2.0: https://www.apache.org/licenses/LICENSE-2.0

.. </legal notes>

parameters
=================

*)

METHOD valueIsMin
VAR_INPUT
	(* current value to check *)
	currentValue	:LTOD;
	(* lower limit for the current value *)
	minimumValue	:LTOD;
	(* message if the assertion is false *)
	message			:AssertMessage;
END_VAR
IF (currentValue < minimumValue) THEN
	THIS^.assertionWasWrong(message, THIS^.getDebugInfo('valueIsMin'));
END_IF
END_METHOD

(*

short summary
=================
This assertion method checks if the current value is not equal to the unexpected value

.. <legal notes>

legal notes
=================
| SPDX-FileCopyrightText: © 2022 ekvip automation GmbH <info@ekvip.de>
| SPDX-License-Identifier: Apache-2.0
| For details check: Apache-2.0_

.. _Apache-2.0: https://www.apache.org/licenses/LICENSE-2.0

.. </legal notes>

parameters
=================

*)

METHOD valueIsNotEqualTo
VAR_INPUT
	(* current value to check *)
	currentValue	:LTOD;
	(* unexpected value to compare *)
	unexpectedValue	:LTOD;
	(* message if the assertion is false *)
	message			:AssertMessage;
END_VAR
IF (currentValue = unexpectedValue) THEN
	THIS^.assertionWasWrong(message, THIS^.getDebugInfo('valueIsNotEqualTo'));
END_IF
END_METHOD

END_FUNCTION_BLOCK

// ---- Assertor/Assertions/FloatAssertions/classes/FloatAssertions.TcPOU
(*

short summary
=================
| This class provides assert statements for floatings (``REAL`` and ``LREAL``)
| It implements :ref:`IFloatAssertions`
| For 32 bit floats (``REAL``) use :ref:`FloatAssertions.single`
| For 64 bit floats (``LREAL``) use :ref:`FloatAssertions.double`

.. <legal notes>

legal notes
=================
| SPDX-FileCopyrightText: © 2022 ekvip automation GmbH <info@ekvip.de>
| SPDX-License-Identifier: Apache-2.0
| For details check: Apache-2.0_

.. _Apache-2.0: https://www.apache.org/licenses/LICENSE-2.0

.. </legal notes>

methods
==================

*)

{attribute 'reflection'}
FUNCTION_BLOCK INTERNAL FloatAssertions EXTENDS CNM_AbstractObject.Object IMPLEMENTS IFloatAssertions, IAssertCallBacksetter
VAR
	(* class to handle assert statements for 32 bit floats *)
	realAssertions	:RealAssertions();
	(* class to handle assert statements for 64 bit floats *)
	lRealAssertions	:LRealAssertions();
END_VAR

(*

short summary
=================
This abstract property returns the class name of the concrete object, 
It's for debugging purpose

.. <legal notes>

legal notes
=================
| SPDX-FileCopyrightText: © 2022 ekvip automation GmbH <info@ekvip.de>
| SPDX-License-Identifier: Apache-2.0
| For details check: Apache-2.0_

.. _Apache-2.0: https://www.apache.org/licenses/LICENSE-2.0

.. </legal notes>

*)

PROPERTY className :CNM_AbstractObject.ClassName
GET
className := 'CNM_AssertionInterfaceLib.FloatAssertions';
END_GET
END_PROPERTY

(*

short summary
=================
Returns the interface :ref:`ILrealAssertions` with assert statements for 64 bit floatings (``LREAL``)

.. <legal notes>

legal notes
=================
| SPDX-FileCopyrightText: © 2022 ekvip automation GmbH <info@ekvip.de>
| SPDX-License-Identifier: Apache-2.0
| For details check: Apache-2.0_

.. _Apache-2.0: https://www.apache.org/licenses/LICENSE-2.0

.. </legal notes>

*)

PROPERTY double :ILrealAssertions
GET
double := THIS^.lrealAssertions;
END_GET
END_PROPERTY

(*

short summary
=================
This methods is the setter for the callback class if an assertion was false

.. <legal notes>

legal notes
=================
| SPDX-FileCopyrightText: © 2022 ekvip automation GmbH <info@ekvip.de>
| SPDX-License-Identifier: Apache-2.0
| For details check: Apache-2.0_

.. _Apache-2.0: https://www.apache.org/licenses/LICENSE-2.0

.. </legal notes>

parameters
=================

*)

METHOD setCallBack
VAR_INPUT
	(* the class that must be informed if an assertion is false *)
	callBack	:IAssertCallback;  
END_VAR
THIS^.realAssertions.setCallBack(callBack);
THIS^.lRealAssertions.setCallBack(callBack);
END_METHOD

(*

short summary
=================
Returns the interface :ref:`IRealAssertions` with assert statements for 32 bit floatings (``REAL``)

.. <legal notes>

legal notes
=================
| SPDX-FileCopyrightText: © 2022 ekvip automation GmbH <info@ekvip.de>
| SPDX-License-Identifier: Apache-2.0
| For details check: Apache-2.0_

.. _Apache-2.0: https://www.apache.org/licenses/LICENSE-2.0

.. </legal notes>

*)

PROPERTY single :IRealAssertions
GET
single := THIS^.realAssertions;
END_GET
END_PROPERTY

END_FUNCTION_BLOCK

// ---- Assertor/Assertions/FloatAssertions/Real/classes/RealAssertions.TcPOU
(*

short summary
=================
This class provides assert statements for 32 bit floatings (``REAL``).
It implements the interface :ref:`IRealAssertions`

.. <legal notes>

legal notes
=================
| SPDX-FileCopyrightText: © 2022 ekvip automation GmbH <info@ekvip.de>
| SPDX-License-Identifier: Apache-2.0
| For details check: Apache-2.0_

.. _Apache-2.0: https://www.apache.org/licenses/LICENSE-2.0

.. </legal notes>

methods
==================

*)

{attribute 'reflection'}
FUNCTION_BLOCK INTERNAL RealAssertions EXTENDS AbstactAssertion IMPLEMENTS IRealAssertions
VAR
END_VAR
VAR CONSTANT
	(* mask for determining value as a special value *)
	MASK_FOR_EXPONENT 	:DWORD := 16#7F80_0000;
	(* mask for determining a special value as NaN or infinite *)  
	MASK_FOR_FRACTION	:DWORD := 16#007F_FFFF;
	(* mask to get the sign bit of an infinite or zero value *)
	MASK_FOR_SIGN_BIT	:DWORD := 16#8000_0000;
	(* just to compare results or the memory of a float value *)
	ZERO				:DWORD := 16#0000_0000;
END_VAR

(*

short summary
=================
This abstract property returns the class name of the concrete object, 
It's for debugging purpose

.. <legal notes>

legal notes
=================
| SPDX-FileCopyrightText: © 2022 ekvip automation GmbH <info@ekvip.de>
| SPDX-License-Identifier: Apache-2.0
| For details check: Apache-2.0_

.. _Apache-2.0: https://www.apache.org/licenses/LICENSE-2.0

.. </legal notes>

*)

PROPERTY className :CNM_AbstractObject.ClassName
GET
className := 'CNM_AssertionInterfaceLib.RealAssertions';
END_GET
END_PROPERTY

(*

short summary
=================
This method checks if a value is infinite
(infinty OR -inifinity), for details check `IEEE 754`_

.. _IEEE 754: https://en.wikipedia.org/wiki/IEEE_754

.. <legal notes>

legal notes
=================
| SPDX-FileCopyrightText: © 2023 ekvip automation GmbH <info@ekvip.de>
| SPDX-License-Identifier: Apache-2.0
| For details check: Apache-2.0_

.. _Apache-2.0: https://www.apache.org/licenses/LICENSE-2.0

.. </legal notes>

parameters
=================
:return: 
``TRUE``: value is inifinty or -infinity
``FALSE``: value is not inifinty and not -infinity

*)

METHOD PROTECTED isValueInfinite :BOOL
VAR_INPUT
	(* value to check *)
	value			:REAL;	
END_VAR
VAR
	(* just to cast the value*)
	realAsDword		:POINTER TO DWORD;
END_VAR
realAsDword := ADR(value);
isValueInfinite := (
	THIS^.isValueSpecial(value)
	AND ((realAsDword^ AND THIS^.MASK_FOR_FRACTION) = THIS^.ZERO)
);
END_METHOD

(*

short summary
=================
This method checks if a value is not a number
(NaN), for details check `IEEE 754`_

.. _IEEE 754: https://en.wikipedia.org/wiki/IEEE_754

.. <legal notes>

legal notes
=================
| SPDX-FileCopyrightText: © 2023 ekvip automation GmbH <info@ekvip.de>
| SPDX-License-Identifier: Apache-2.0
| For details check: Apache-2.0_

.. _Apache-2.0: https://www.apache.org/licenses/LICENSE-2.0

.. </legal notes>

parameters
=================
:return: 
``TRUE``: value is NaN
``FALSE``: value is not NaN

*)

METHOD PROTECTED isValueNaN :BOOL
VAR_INPUT
	(* value to check *)
	value			:REAL;	
END_VAR
VAR
	(* just to cast the value*)
	realAsDword		:POINTER TO DWORD;
END_VAR
realAsDword := ADR(value);
isValueNaN := (
	THIS^.isValueSpecial(value)
	AND ((realAsDword^ AND THIS^.MASK_FOR_FRACTION) > THIS^.ZERO)
);
END_METHOD

(*

short summary
=================
This method checks if a value is negative infinite
(-inifinity), for details check `IEEE 754`_

.. _IEEE 754: https://en.wikipedia.org/wiki/IEEE_754

.. <legal notes>

legal notes
=================
| SPDX-FileCopyrightText: © 2023 ekvip automation GmbH <info@ekvip.de>
| SPDX-License-Identifier: Apache-2.0
| For details check: Apache-2.0_

.. _Apache-2.0: https://www.apache.org/licenses/LICENSE-2.0

.. </legal notes>

parameters
=================
:return: 
``TRUE``: value is -infinity
``FALSE``: value is not -infinity

*)

METHOD PROTECTED isValueNegativeInfinite : BOOL
VAR_INPUT
	(* value to check *)
	value			:REAL;	
END_VAR
VAR
	(* just to cast the value*)
	realAsDword		:POINTER TO DWORD;
END_VAR
realAsDword := ADR(value);
isValueNegativeInfinite := (
	THIS^.isValueInfinite(value)
	AND ((realAsDword^ AND THIS^.MASK_FOR_SIGN_BIT) = THIS^.MASK_FOR_SIGN_BIT)
);
END_METHOD

(*

short summary
=================
This method checks if a value is positive infinite
(infinty), for details check `IEEE 754`_

.. _IEEE 754: https://en.wikipedia.org/wiki/IEEE_754

.. <legal notes>

legal notes
=================
| SPDX-FileCopyrightText: © 2023 ekvip automation GmbH <info@ekvip.de>
| SPDX-License-Identifier: Apache-2.0
| For details check: Apache-2.0_

.. _Apache-2.0: https://www.apache.org/licenses/LICENSE-2.0

.. </legal notes>

parameters
=================
:return: 
``TRUE``: value is inifinty
``FALSE``: value is not inifinty

*)

METHOD PROTECTED isValuePositiveInfinite :BOOL
VAR_INPUT
	(* value to check *)
	value			:REAL;	
END_VAR
VAR
	(* just to cast the value*)
	realAsDword		:POINTER TO DWORD;
END_VAR
realAsDword := ADR(value);
isValuePositiveInfinite := (
	THIS^.isValueInfinite(value)
	AND ((realAsDword^ AND THIS^.MASK_FOR_SIGN_BIT) = THIS^.ZERO)
);
END_METHOD

(*

short summary
=================
This method checks if a value is a special value
(NaN OR infinty OR -inifinity), for details check `IEEE 754`_

.. _IEEE 754: https://en.wikipedia.org/wiki/IEEE_754

.. <legal notes>

legal notes
=================
| SPDX-FileCopyrightText: © 2023 ekvip automation GmbH <info@ekvip.de>
| SPDX-License-Identifier: Apache-2.0
| For details check: Apache-2.0_

.. _Apache-2.0: https://www.apache.org/licenses/LICENSE-2.0

.. </legal notes>

parameters
=================
:return: 
``TRUE``: value is inifinty or -infinity or NaN
``FALSE``: value is not inifinty and not -infinity and not NaN

*)

METHOD PROTECTED isValueSpecial :BOOL
VAR_INPUT
	(* value to check *)
	value			:REAL;	
END_VAR
VAR
	(* just to cast the value*)
	realAsDword		:POINTER TO DWORD;
END_VAR
realAsDword := ADR(value);
isValueSpecial := ((realAsDword^ AND THIS^.MASK_FOR_EXPONENT) = THIS^.MASK_FOR_EXPONENT);
END_METHOD

(*

short summary
=================
This assertion method checks if the current value is a number (NOT NaN)
for details check `IEEE 754`_

.. _IEEE 754: https://en.wikipedia.org/wiki/IEEE_754

.. <legal notes>

legal notes
=================
| SPDX-FileCopyrightText: © 2023 ekvip automation GmbH <info@ekvip.de>
| SPDX-License-Identifier: Apache-2.0
| For details check: Apache-2.0_

.. _Apache-2.0: https://www.apache.org/licenses/LICENSE-2.0

.. </legal notes>

parameters
=================

*)

METHOD valueIsANumber
VAR_INPUT
	(* current value to check *)
	currentValue	:REAL;
	(* message if the assertion is false *)
	message			:AssertMessage;
END_VAR
IF (THIS^.isValueNaN(currentValue)) THEN
	THIS^.assertionWasWrong(message, THIS^.getDebugInfo('valueIsANumber'));
END_IF
END_METHOD

(*

short summary
=================
This assertion method checks if the current value is equal to the expected value

.. attention:: 
	Nothing is equal to NaN, that means if ``currentValue`` OR ``expectedValue`` OR ``tolerance``
	is NaN then is the assertion false. For details check `IEEE 754`_

.. attention:: 
	infinity is equal to infinity and -infinity is equal to -infinity, that means if
	``currentValue`` AND ``expectedValue`` have the value infinity 
	OR ``currentValue`` AND ``expectedValue`` have the value -infinity
	the assertion is TRUE. For details check `IEEE 754`_

.. attention:: 
	If ``tolerance`` has the value infinity or -infinity and 
	``currentValue`` is not NaN and ``expectedValue`` is not NaN
	then is the assertion true. For details check `IEEE 754`_

.. _IEEE 754: https://en.wikipedia.org/wiki/IEEE_754

.. <legal notes>

legal notes
=================
| SPDX-FileCopyrightText: © 2022 ekvip automation GmbH <info@ekvip.de>
| SPDX-License-Identifier: Apache-2.0
| For details check: Apache-2.0_

.. _Apache-2.0: https://www.apache.org/licenses/LICENSE-2.0

.. </legal notes>

parameters
=================

*)

METHOD valueIsEqualTo
VAR_INPUT
	(* current value to check *)
	currentValue	:REAL;
	(* expected value to compare *)
	expectedValue	:REAL;
	(* tolerance to compensate twiddling floats, it has no sign *)
	tolerance		:REAL;
	(* message if the assertion is false *)
	message			:AssertMessage;
END_VAR
IF (
	THIS^.isValueNaN(currentValue)
	OR THIS^.isValueNaN(expectedValue)
	OR THIS^.isValueNaN(tolerance)
) THEN
	THIS^.assertionWasWrong(message, THIS^.getDebugInfo('valueIsEqualTo'));
ELSIF (THIS^.isValueInfinite(tolerance)) THEN
	RETURN;
ELSIF (
	THIS^.isValueInfinite(currentValue)
	OR THIS^.isValueInfinite(expectedValue)
	OR THIS^.isValueInfinite(tolerance)
) THEN
	RETURN (THIS^.isValuePositiveInfinite(currentValue) AND THIS^.isValuePositiveInfinite(expectedValue));
	RETURN (THIS^.isValueNegativeInfinite(currentValue) AND THIS^.isValueNegativeInfinite(expectedValue));
	THIS^.assertionWasWrong(message, THIS^.getDebugInfo('valueIsEqualTo'));	
ELSIF (ABS(currentValue-expectedValue) > ABS(tolerance)) THEN
	THIS^.assertionWasWrong(message, THIS^.getDebugInfo('valueIsEqualTo'));
END_IF
END_METHOD

(*

short summary
=================
This assertion method checks if the current value is finite
(NOT (infinty OR -inifinity)), for details check `IEEE 754`_

.. _IEEE 754: https://en.wikipedia.org/wiki/IEEE_754

.. <legal notes>

legal notes
=================
| SPDX-FileCopyrightText: © 2023 ekvip automation GmbH <info@ekvip.de>
| SPDX-License-Identifier: Apache-2.0
| For details check: Apache-2.0_

.. _Apache-2.0: https://www.apache.org/licenses/LICENSE-2.0

.. </legal notes>

parameters
=================

*)

METHOD valueIsFinite
VAR_INPUT
	(* current value to check *)
	currentValue	:REAL;
	(* message if the assertion is false *)
	message			:AssertMessage;
END_VAR
IF (THIS^.isValueInfinite(currentValue)) THEN
	THIS^.assertionWasWrong(message, THIS^.getDebugInfo('valueIsFinite'));
END_IF
END_METHOD

(*

short summary
=================
This assertion method checks if the current value is greater than the less value

.. attention:: 
	Any comparsion to NaN is ``FALSE`` that means if ``currentValue`` OR ``lessValue``
	is NaN then is the assertion false.
	For details check `IEEE 754`_ and the truth table below.

.. attention:: 
	Every number is smaller than infinity except -infinity, it's equal.
	Every number is greater than -infinity except -infinity, it's equal.
	For details check `IEEE 754`_ and the truth table below.

.. _IEEE 754: https://en.wikipedia.org/wiki/IEEE_754

truth table for special values
===============================
+----------------------+-------------------+---------------+
| **``currentValue``** | **``lessValue``** | **assertion** |
+======================+===================+===============+
| NaN                  | Any value         | FASLE         |
+----------------------+-------------------+---------------+
| Any value            | NaN               | FALSE         |
+----------------------+-------------------+---------------+
| infinity             | NOT NaN           | TRUE          |
|                      | NOT infinity      |               |
+----------------------+-------------------+---------------+
| -infinty             | Any value         | FALSE         |
+----------------------+-------------------+---------------+
| Any value            | infinity          | FALSE         |
+----------------------+-------------------+---------------+
| NOT NaN              | -inifinity        | TRUE          |
| NOT -infinity        |                   |               |
+----------------------+-------------------+---------------+

.. <legal notes>

legal notes
=================
| SPDX-FileCopyrightText: © 2022 ekvip automation GmbH <info@ekvip.de>
| SPDX-License-Identifier: Apache-2.0
| For details check: Apache-2.0_

.. _Apache-2.0: https://www.apache.org/licenses/LICENSE-2.0

.. </legal notes>

parameters
=================

*)

METHOD valueIsGreaterThan
VAR_INPUT
	(* current value to check *)
	currentValue	:REAL;
	(* less than lower limit *)
	lessValue		:REAL;
	(* message if the assertion is false *)
	message			:AssertMessage;
END_VAR
IF (THIS^.isValueNaN(currentValue) OR THIS^.isValueNaN(lessValue)) THEN
	THIS^.assertionWasWrong(message, THIS^.getDebugInfo('valueIsGreaterThan'));
ELSIF (THIS^.isValueNegativeInfinite(currentValue)) THEN
	THIS^.assertionWasWrong(message, THIS^.getDebugInfo('valueIsGreaterThan'));
ELSIF (THIS^.isValuePositiveInfinite(lessValue)) THEN
	THIS^.assertionWasWrong(message, THIS^.getDebugInfo('valueIsGreaterThan'));
ELSIF (THIS^.isValueNegativeInfinite(lessValue)) THEN
	RETURN;
ELSIF (THIS^.isValuePositiveInfinite(currentValue)) THEN
	RETURN;
ELSIF (currentValue <= lessValue) THEN
	THIS^.assertionWasWrong(message, THIS^.getDebugInfo('valueIsGreaterThan'));
END_IF
END_METHOD

(*

short summary
=================
This assertion method checks if the current value is infinite
(infinty OR -inifinity), for details check `IEEE 754`_

.. _IEEE 754: https://en.wikipedia.org/wiki/IEEE_754

.. <legal notes>

legal notes
=================
| SPDX-FileCopyrightText: © 2023 ekvip automation GmbH <info@ekvip.de>
| SPDX-License-Identifier: Apache-2.0
| For details check: Apache-2.0_

.. _Apache-2.0: https://www.apache.org/licenses/LICENSE-2.0

.. </legal notes>

parameters
=================

*)

METHOD valueIsInfinite
VAR_INPUT
	(* current value to check *)
	currentValue	:REAL;
	(* message if the assertion is false *)
	message			:AssertMessage;
END_VAR
IF (NOT THIS^.isValueInfinite(currentValue)) THEN
	THIS^.assertionWasWrong(message, THIS^.getDebugInfo('valueIsInfinite'));
END_IF
END_METHOD

(*

short summary
=================
This assertion method checks if the current value is inside a limit

.. attention:: 
	limits are included: ``valueIsInRangeOf(3.0, 3.0, 3.0)`` is a true assertion

.. attention:: 
	Any comparsion to NaN is ``FALSE`` that means 
	if ``lowerLimit`` OR ``currentValue`` OR ``upperLimit``
	is NaN then is the assertion false.
	For details check `IEEE 754`_ and the truth table below.

.. attention:: 
	Every number is smaller than infinity except -infinity, it's equal.
	Every number is greater than -infinity except -infinity, it's equal.
	For details check `IEEE 754`_ and the truth table below.

.. _IEEE 754: https://en.wikipedia.org/wiki/IEEE_754

truth table for special values
===============================
+--------------------+----------------------+--------------------+---------------+
| **``lowerLimit``** | **``currentValue``** | **``upperLimit``** | **assertion** |
+====================+======================+====================+===============+
| NaN                | Any value            | Any value          | FASLE         |
+--------------------+----------------------+--------------------+---------------+
| Any value          | NaN                  | Any value          | FALSE         |
+--------------------+----------------------+--------------------+---------------+
| Any value          | Any value            | NaN                | FALSE         |
+--------------------+----------------------+--------------------+---------------+
| -infinity          | NOT NaN              | infinity           | TRUE          |
+--------------------+----------------------+--------------------+---------------+
| infinity           | Any value            | -infinity          | FALSE         |
+--------------------+----------------------+--------------------+---------------+
| NOT -infinity      | -infinity            | Any value          | FALSE         |
+--------------------+----------------------+--------------------+---------------+
| Any value          | infinity             | NOT infinity       | FALSE         |
+--------------------+----------------------+--------------------+---------------+
| -infinity          | -infinity            | -infinity          | TRUE          |
+--------------------+----------------------+--------------------+---------------+
| infinity           | infinity             | infinity           | TRUE          |
+--------------------+----------------------+--------------------+---------------+
| -infinity          | NOT -infinity        | -infinity          | FALSE         |
+--------------------+----------------------+--------------------+---------------+
| infinity           | NOT infinity         | infinity           | FALSE         |
+--------------------+----------------------+--------------------+---------------+

.. <legal notes>

legal notes
=================
| SPDX-FileCopyrightText: © 2022 ekvip automation GmbH <info@ekvip.de>
| SPDX-License-Identifier: Apache-2.0
| For details check: Apache-2.0_

.. _Apache-2.0: https://www.apache.org/licenses/LICENSE-2.0

.. </legal notes>

parameters
=================

*)

METHOD valueIsInRangeOf
VAR_INPUT
	(* lower limit for the current value *)
	lowerLimit		:REAL;
	(* current value to check *)
	currentValue	:REAL;
	(* upper limit for the current value *)
	upperLimit		:REAL;
	(* message if the assertion is false *)
	message			:AssertMessage;
END_VAR
IF (THIS^.isValueNaN(lowerLimit) OR THIS^.isValueNaN(currentValue) OR THIS^.isValueNaN(upperLimit)) THEN
	THIS^.assertionWasWrong(message, THIS^.getDebugInfo('valueIsInRangeOf'));
ELSIF (THIS^.isValueNegativeInfinite(upperLimit) AND THIS^.isValuePositiveInfinite(lowerLimit)) THEN	
	THIS^.assertionWasWrong(message, THIS^.getDebugInfo('valueIsInRangeOf'));
ELSIF (THIS^.isValueNegativeInfinite(currentValue) AND (NOT THIS^.isValueNegativeInfinite(lowerLimit))) THEN
	THIS^.assertionWasWrong(message, THIS^.getDebugInfo('valueIsInRangeOf'));
ELSIF (THIS^.isValuePositiveInfinite(currentValue) AND (NOT THIS^.isValuePositiveInfinite(upperLimit))) THEN
	THIS^.assertionWasWrong(message, THIS^.getDebugInfo('valueIsInRangeOf'));
ELSIF (
	THIS^.isValuePositiveInfinite(lowerLimit)
	AND (NOT THIS^.isValuePositiveInfinite(currentValue))
	AND THIS^.isValuePositiveInfinite(upperLimit)
) THEN
	THIS^.assertionWasWrong(message, THIS^.getDebugInfo('valueIsInRangeOf'));
ELSIF (
	THIS^.isValueNegativeInfinite(lowerLimit)
	AND (NOT THIS^.isValueNegativeInfinite(currentValue))
	AND THIS^.isValueNegativeInfinite(upperLimit)
) THEN
	THIS^.assertionWasWrong(message, THIS^.getDebugInfo('valueIsInRangeOf'));
ELSIF (
	THIS^.isValuePositiveInfinite(lowerLimit)
	AND THIS^.isValuePositiveInfinite(currentValue)
	AND THIS^.isValuePositiveInfinite(upperLimit)
) THEN
	RETURN;
ELSIF (
	THIS^.isValueNegativeInfinite(lowerLimit)
	AND THIS^.isValueNegativeInfinite(currentValue)
	AND THIS^.isValueNegativeInfinite(upperLimit)
) THEN
	RETURN;
ELSIF (THIS^.isValueNegativeInfinite(lowerLimit) AND THIS^.isValuePositiveInfinite(upperLimit)) THEN
	RETURN;
ELSIF ((currentValue < lowerLimit) OR (currentValue > upperLimit)) THEN
	THIS^.assertionWasWrong(message, THIS^.getDebugInfo('valueIsInRangeOf'));
END_IF
END_METHOD

(*

short summary
=================
This assertion method checks if the current value is greater than the less value

.. attention::
	Any comparsion to NaN is ``FALSE`` that means if ``currentValue`` OR ``greaterValue``
	is NaN then is the assertion false.
	For details check `IEEE 754`_ and the truth table below.

.. attention::
	Every number is smaller than infinity except -infinity, it's equal.
	Every number is greater than -infinity except -infinity, it's equal.
	For details check `IEEE 754`_ and the truth table below.

.. _IEEE 754: https://en.wikipedia.org/wiki/IEEE_754

truth table for special values
===============================
+----------------------+----------------------+---------------+
| **``currentValue``** | **``greaterValue``** | **assertion** |
+======================+======================+===============+
| NaN                  | Any value            | FASLE         |
+----------------------+----------------------+---------------+
| Any value            | NaN                  | FALSE         |
+----------------------+----------------------+---------------+
| infinity             | Any value            | FALSE         |
+----------------------+----------------------+---------------+
| -infinty             | NOT NaN              | TRUE          |
|                      | NOT -infinity        |               |
+----------------------+----------------------+---------------+
| NOT NaN              | infinity             | TRUE          |
| NOT infinity         |                      |               |
+----------------------+----------------------+---------------+

.. <legal notes>

legal notes
=================
| SPDX-FileCopyrightText: © 2022 ekvip automation GmbH <info@ekvip.de>
| SPDX-License-Identifier: Apache-2.0
| For details check: Apache-2.0_

.. _Apache-2.0: https://www.apache.org/licenses/LICENSE-2.0

.. </legal notes>

parameters
=================

*)

METHOD valueIsLessThan
VAR_INPUT
	(* current value to check *)
	currentValue	:REAL;
	(* greater than upper limit *)
	greaterValue	:REAL;
	(* message if the assertion is false *)
	message			:AssertMessage;
END_VAR
IF (THIS^.isValueNaN(currentValue) OR THIS^.isValueNaN(greaterValue)) THEN
	THIS^.assertionWasWrong(message, THIS^.getDebugInfo('valueIsLessThan'));
ELSIF (THIS^.isValuePositiveInfinite(currentValue)) THEN
	THIS^.assertionWasWrong(message, THIS^.getDebugInfo('valueIsLessThan'));
ELSIF (THIS^.isValueNegativeInfinite(greaterValue)) THEN
	THIS^.assertionWasWrong(message, THIS^.getDebugInfo('valueIsLessThan'));
ELSIF (THIS^.isValuePositiveInfinite(greaterValue)) THEN
	RETURN;
ELSIF (THIS^.isValueNegativeInfinite(currentValue)) THEN
	RETURN;
ELSIF (currentValue >= greaterValue) THEN
	THIS^.assertionWasWrong(message, THIS^.getDebugInfo('valueIsLessThan'));
END_IF
END_METHOD

(*

short summary
=================
This assertion method checks if the current value is less than or equal to the maximum value

.. attention::
	Any comparsion to NaN is ``FALSE`` that means if ``currentValue`` OR ``maximumValue``
	is NaN then is the assertion false.
	For details check `IEEE 754`_ and the truth table below.

.. attention::
	Every number is smaller than infinity except -infinity, it's equal.
	Every number is greater than -infinity except -infinity, it's equal.
	For details check `IEEE 754`_ and the truth table below.

.. _IEEE 754: https://en.wikipedia.org/wiki/IEEE_754

truth table for special values
===============================
+----------------------+----------------------+---------------+
| **``currentValue``** | **``maximumValue``** | **assertion** |
+======================+======================+===============+
| NaN                  | Any value            | FASLE         |
+----------------------+----------------------+---------------+
| Any value            | NaN                  | FALSE         |
+----------------------+----------------------+---------------+
| NOT NaN              | infinity             | TRUE          |
+----------------------+----------------------+---------------+
| -infinity            | NOT NaN              | TRUE          |
+----------------------+----------------------+---------------+
| infinity             | NOT infinity         | FALSE         |
+----------------------+----------------------+---------------+
| NOT -infinity        | -infinity            | FALSE         |
+----------------------+----------------------+---------------+

.. <legal notes>

legal notes
=================
| SPDX-FileCopyrightText: © 2022 ekvip automation GmbH <info@ekvip.de>
| SPDX-License-Identifier: Apache-2.0
| For details check: Apache-2.0_

.. _Apache-2.0: https://www.apache.org/licenses/LICENSE-2.0

.. </legal notes>

parameters
=================

*)

METHOD valueIsMax
VAR_INPUT
	(* current value to check *)
	currentValue	:REAL;
	(* upper limit for the current value *)
	maximumValue	:REAL;
	(* message if the assertion is false *)
	message			:AssertMessage;
END_VAR
IF (THIS^.isValueNaN(currentValue) OR THIS^.isValueNaN(maximumValue)) THEN
	THIS^.assertionWasWrong(message, THIS^.getDebugInfo('valueIsMax'));
ELSIF (
	THIS^.isValueNegativeInfinite(maximumValue)
	AND (NOT THIS^.isValueNegativeInfinite(currentValue))
) THEN
	THIS^.assertionWasWrong(message, THIS^.getDebugInfo('valueIsMax'));
ELSIF (
	THIS^.isValuePositiveInfinite(currentValue)
	AND (NOT THIS^.isValuePositiveInfinite(maximumValue))
) THEN
	THIS^.assertionWasWrong(message, THIS^.getDebugInfo('valueIsMax'));
ELSIF (THIS^.isValuePositiveInfinite(maximumValue)) THEN
	RETURN;	
ELSIF (THIS^.isValueNegativeInfinite(currentValue)) THEN
	RETURN;
ELSIF (currentValue > maximumValue) THEN
	THIS^.assertionWasWrong(message, THIS^.getDebugInfo('valueIsMax'));
END_IF
END_METHOD

(*

short summary
=================
This assertion method checks if the current value is greater than or equal to the minimum value

.. attention::
	Any comparsion to NaN is ``FALSE`` that means if ``currentValue`` OR ``minimumValue``
	is NaN then is the assertion false.
	For details check `IEEE 754`_ and the truth table below.

.. attention::
	Every number is smaller than infinity except -infinity, it's equal.
	Every number is greater than -infinity except -infinity, it's equal.
	For details check `IEEE 754`_ and the truth table below.

.. _IEEE 754: https://en.wikipedia.org/wiki/IEEE_754

truth table for special values
===============================
+----------------------+----------------------+---------------+
| **``currentValue``** | **``minimumValue``** | **assertion** |
+======================+======================+===============+
| NaN                  | Any value            | FASLE         |
+----------------------+----------------------+---------------+
| Any value            | NaN                  | FALSE         |
+----------------------+----------------------+---------------+
| infinity             | NOT NaN              | TRUE          |
+----------------------+----------------------+---------------+
| NOT NaN              | -infinity            | TRUE          |
+----------------------+----------------------+---------------+
| -infinity            | NOT -infinity        | FALSE         |
+----------------------+----------------------+---------------+
| NOT infinity         | infinity             | FALSE         |
+----------------------+----------------------+---------------+

.. <legal notes>

legal notes
=================
| SPDX-FileCopyrightText: © 2022 ekvip automation GmbH <info@ekvip.de>
| SPDX-License-Identifier: Apache-2.0
| For details check: Apache-2.0_

.. _Apache-2.0: https://www.apache.org/licenses/LICENSE-2.0

.. </legal notes>

parameters
=================

*)

METHOD valueIsMin
VAR_INPUT
	(* current value to check *)
	currentValue	:REAL;
	(* lower limit for the current value *)
	minimumValue	:REAL;
	(* message if the assertion is false *)
	message			:AssertMessage;
END_VAR
IF (THIS^.isValueNaN(currentValue) OR THIS^.isValueNaN(minimumValue)) THEN
	THIS^.assertionWasWrong(message, THIS^.getDebugInfo('valueIsMin'));
ELSIF (
	THIS^.isValueNegativeInfinite(currentValue)
	AND (NOT THIS^.isValueNegativeInfinite(minimumValue))
) THEN
	THIS^.assertionWasWrong(message, THIS^.getDebugInfo('valueIsMin'));
ELSIF (
	THIS^.isValuePositiveInfinite(minimumValue)
	AND (NOT THIS^.isValuePositiveInfinite(currentValue))
) THEN
	THIS^.assertionWasWrong(message, THIS^.getDebugInfo('valueIsMin'));
ELSIF (THIS^.isValuePositiveInfinite(currentValue)) THEN
	RETURN;	
ELSIF (THIS^.isValueNegativeInfinite(minimumValue)) THEN
	RETURN;
ELSIF (currentValue < minimumValue) THEN
	THIS^.assertionWasWrong(message, THIS^.getDebugInfo('valueIsMin'));
END_IF
END_METHOD

(*

short summary
=================
This assertion method checks if the current value is a not a number (NaN)
for details check `IEEE 754`_

.. _IEEE 754: https://en.wikipedia.org/wiki/IEEE_754

.. <legal notes>

legal notes
=================
| SPDX-FileCopyrightText: © 2023 ekvip automation GmbH <info@ekvip.de>
| SPDX-License-Identifier: Apache-2.0
| For details check: Apache-2.0_

.. _Apache-2.0: https://www.apache.org/licenses/LICENSE-2.0

.. </legal notes>

parameters
=================

*)

METHOD valueIsNaN
VAR_INPUT
	(* current value to check *)
	currentValue	:REAL;
	(* message if the assertion is false *)
	message			:AssertMessage;
END_VAR
IF (NOT THIS^.isValueNaN(currentValue)) THEN
	THIS^.assertionWasWrong(message, THIS^.getDebugInfo('valueIsNaN'));
END_IF
END_METHOD

(*

short summary
=================
This assertion method checks if the current value is negative

.. attention::
	Any comparsion to NaN is ``FALSE`` that means if ``currentValue``
	is NaN then is the assertion false.
	For details check `IEEE 754`_.

.. attention::
	``currentValue`` has the value infinity means the assertion is false.
	``currentValue`` has the value -infinity means the assertion is true.
	``currentValue`` has the +0.0 means the assertion is false.
	``currentValue`` has the value -0.0 means the assertion is true.	
	For details check `IEEE 754`_.

.. _IEEE 754: https://en.wikipedia.org/wiki/IEEE_754

.. <legal notes>

legal notes
=================
| SPDX-FileCopyrightText: © 2022 ekvip automation GmbH <info@ekvip.de>
| SPDX-License-Identifier: Apache-2.0
| For details check: Apache-2.0_

.. _Apache-2.0: https://www.apache.org/licenses/LICENSE-2.0

.. </legal notes>

parameters
=================

*)

METHOD valueIsNegative
VAR_INPUT
	(* current value to check *)
	currentValue	:REAL;
	(* message if the assertion is false *)
	message			:AssertMessage;
END_VAR
VAR
	(* just to cast ``currentValue`` *)
	currentValueAsDWord	:POINTER TO DWORD;
END_VAR
IF (THIS^.isValueNaN(currentValue)) THEN	
	THIS^.assertionWasWrong(message, THIS^.getDebugInfo('valueIsNegative'));
ELSE
	currentValueAsDWord := ADR(currentValue);
	IF ((currentValueAsDWord^ AND THIS^.MASK_FOR_SIGN_BIT) = THIS^.ZERO) THEN
		THIS^.assertionWasWrong(message, THIS^.getDebugInfo('valueIsNegative'));
	END_IF
END_IF
END_METHOD

(*

short summary
=================
This assertion method checks if the current value is negative infinite
(-infinty), for details check `IEEE 754`_

.. _IEEE 754: https://en.wikipedia.org/wiki/IEEE_754

.. <legal notes>

legal notes
=================
| SPDX-FileCopyrightText: © 2023 ekvip automation GmbH <info@ekvip.de>
| SPDX-License-Identifier: Apache-2.0
| For details check: Apache-2.0_

.. _Apache-2.0: https://www.apache.org/licenses/LICENSE-2.0

.. </legal notes>

parameters
=================

*)

METHOD valueIsNegativeInfinite
VAR_INPUT
	(* current value to check *)
	currentValue	:REAL;
	(* message if the assertion is false *)
	message			:AssertMessage;
END_VAR
IF (NOT THIS^.isValueNegativeInfinite(currentValue)) THEN
	THIS^.assertionWasWrong(message, THIS^.getDebugInfo('valueIsNegativeInfinite'));
END_IF
END_METHOD

(*

short summary
=================
This assertion method checks if the current value is +0.0
for details check `IEEE 754`_

.. _IEEE 754: https://en.wikipedia.org/wiki/IEEE_754

.. <legal notes>

legal notes
=================
| SPDX-FileCopyrightText: © 2023 ekvip automation GmbH <info@ekvip.de>
| SPDX-License-Identifier: Apache-2.0
| For details check: Apache-2.0_

.. _Apache-2.0: https://www.apache.org/licenses/LICENSE-2.0

.. </legal notes>

parameters
=================

*)

METHOD valueIsNegativeZero
VAR_INPUT
	(* current value to check *)
	currentValue	:REAL;
	(* message if the assertion is false *)
	message			:AssertMessage;
END_VAR
VAR
	(* just to cast ``currentValue`` *)
	currentValueAsDWord	:POINTER TO DWORD;
END_VAR
currentValueAsDWord := ADR(currentValue);
IF (currentValueAsDWord^ <> THIS^.MASK_FOR_SIGN_BIT) THEN
	THIS^.assertionWasWrong(message, THIS^.getDebugInfo('valueIsNegativeZero'));
END_IF
END_METHOD

(*

short summary
=================
This assertion method checks if the current value is a normal number
(a finite non-zero/non-subnormal floating-point number)
for details check `IEEE 754`_

.. _IEEE 754: https://en.wikipedia.org/wiki/IEEE_754

.. <legal notes>

legal notes
=================
| SPDX-FileCopyrightText: © 2023 ekvip automation GmbH <info@ekvip.de>
| SPDX-License-Identifier: Apache-2.0
| For details check: Apache-2.0_

.. _Apache-2.0: https://www.apache.org/licenses/LICENSE-2.0

.. </legal notes>

parameters
=================

*)

METHOD valueIsNormal
VAR_INPUT
	(* current value to check *)
	currentValue	:REAL;
	(* message if the assertion is false *)
	message			:AssertMessage;
END_VAR
VAR
	(* just to cast ``currentValue`` *)
	currentValueAsDWord	:POINTER TO DWORD;
END_VAR
IF (THIS^.isValueNaN(currentValue) OR THIS^.isValueInfinite(currentValue)) THEN
	THIS^.assertionWasWrong(message, THIS^.getDebugInfo('valueIsNormal'));
ELSE
	currentValueAsDWord := ADR(currentValue);
	IF ((currentValueAsDWord^ AND THIS^.MASK_FOR_EXPONENT) = THIS^.ZERO) THEN
		THIS^.assertionWasWrong(message, THIS^.getDebugInfo('valueIsNormal'));
	END_IF
END_IF
END_METHOD

(*

short summary
=================
This assertion method checks if the current value is not equal to the unexpected value

.. attention:: 
	Nothing is equal to NaN, that means if ``currentValue`` OR ``unexpectedValue`` OR ``tolerance``
	is NaN then is the assertion true. For details check `IEEE 754`_

.. attention:: 
	infinity is equal to infinity and -infinity is equal to -infinity, that means if
	``currentValue`` AND ``unexpectedValue`` have the value infinity 
	OR ``currentValue`` AND ``unexpectedValue`` have the value -infinity
	the assertion is false. For details check `IEEE 754`_

.. attention:: 
	If ``tolerance`` has the value infinity or -infinity and 
	``currentValue`` is not NaN and ``unexpectedValue`` is not NaN
	then is the assertion false. For details check `IEEE 754`_

.. _IEEE 754: https://en.wikipedia.org/wiki/IEEE_754

.. <legal notes>

legal notes
=================
| SPDX-FileCopyrightText: © 2022 ekvip automation GmbH <info@ekvip.de>
| SPDX-License-Identifier: Apache-2.0
| For details check: Apache-2.0_

.. _Apache-2.0: https://www.apache.org/licenses/LICENSE-2.0

.. </legal notes>

parameters
=================

*)

METHOD valueIsNotEqualTo
VAR_INPUT
	(* current value to check *)
	currentValue	:REAL;
	(* unexpected value to compare *)
	unexpectedValue	:REAL;
	(* tolerance to compensate twiddling floats, it has no sign *)
	tolerance		:REAL;
	(* message if the assertion is false *)
	message			:AssertMessage;
END_VAR
IF (
	THIS^.isValueNaN(currentValue)
	OR THIS^.isValueNaN(unexpectedValue)
	OR THIS^.isValueNaN(tolerance)
) THEN
	RETURN;
ELSIF (THIS^.isValueInfinite(tolerance)) THEN
	THIS^.assertionWasWrong(message, THIS^.getDebugInfo('valueIsNotEqualTo'));
ELSIF (
	THIS^.isValueInfinite(currentValue)
	OR THIS^.isValueInfinite(unexpectedValue)
) THEN
	RETURN (THIS^.isValuePositiveInfinite(currentValue) AND (NOT THIS^.isValuePositiveInfinite(unexpectedValue)));
	RETURN (THIS^.isValueNegativeInfinite(currentValue) AND (NOT THIS^.isValueNegativeInfinite(unexpectedValue)));
	RETURN (THIS^.isValuePositiveInfinite(unexpectedValue) AND (NOT THIS^.isValuePositiveInfinite(currentValue)));
	RETURN (THIS^.isValueNegativeInfinite(unexpectedValue) AND (NOT THIS^.isValueNegativeInfinite(currentValue)));
	THIS^.assertionWasWrong(message, THIS^.getDebugInfo('valueIsNotEqualTo'));
ELSIF (ABS(currentValue-unexpectedValue) <= ABS(tolerance)) THEN
	THIS^.assertionWasWrong(message, THIS^.getDebugInfo('valueIsNotEqualTo'));
END_IF
END_METHOD

(*

short summary
=================
This assertion method checks if the current value is not negative infinite
NOT (-infinty), for details check `IEEE 754`_

.. _IEEE 754: https://en.wikipedia.org/wiki/IEEE_754

.. <legal notes>

legal notes
=================
| SPDX-FileCopyrightText: © 2023 ekvip automation GmbH <info@ekvip.de>
| SPDX-License-Identifier: Apache-2.0
| For details check: Apache-2.0_

.. _Apache-2.0: https://www.apache.org/licenses/LICENSE-2.0

.. </legal notes>

parameters
=================

*)

METHOD valueIsNotNegativeInfinite
VAR_INPUT
	(* current value to check *)
	currentValue	:REAL;
	(* message if the assertion is false *)
	message			:AssertMessage;
END_VAR
IF (THIS^.isValueNegativeInfinite(currentValue)) THEN
	THIS^.assertionWasWrong(message, THIS^.getDebugInfo('valueIsNotNegativeInfinite'));
END_IF
END_METHOD

(*

short summary
=================
This assertion method checks if the current value is not positive infinite
NOT (infinty), for details check `IEEE 754`_

.. _IEEE 754: https://en.wikipedia.org/wiki/IEEE_754

.. <legal notes>

legal notes
=================
| SPDX-FileCopyrightText: © 2023 ekvip automation GmbH <info@ekvip.de>
| SPDX-License-Identifier: Apache-2.0
| For details check: Apache-2.0_

.. _Apache-2.0: https://www.apache.org/licenses/LICENSE-2.0

.. </legal notes>

parameters
=================

*)

METHOD valueIsNotPositiveInfinite
VAR_INPUT
	(* current value to check *)
	currentValue	:REAL;
	(* message if the assertion is false *)
	message			:AssertMessage;
END_VAR
IF (THIS^.isValuePositiveInfinite(currentValue)) THEN
	THIS^.assertionWasWrong(message, THIS^.getDebugInfo('valueIsNotPositiveInfinite'));
END_IF
END_METHOD

(*

short summary
=================
This assertion method checks if the current value is a non special number
(NOT (NaN OR infinty OR -inifinity)), for details check `IEEE 754`_

.. _IEEE 754: https://en.wikipedia.org/wiki/IEEE_754

.. <legal notes>

legal notes
=================
| SPDX-FileCopyrightText: © 2023 ekvip automation GmbH <info@ekvip.de>
| SPDX-License-Identifier: Apache-2.0
| For details check: Apache-2.0_

.. _Apache-2.0: https://www.apache.org/licenses/LICENSE-2.0

.. </legal notes>

parameters
=================

*)

METHOD valueIsNotSpecial : BOOL
VAR_INPUT
	(* current value to check *)
	currentValue	:REAL;
	(* message if the assertion is false *)
	message			:AssertMessage;
END_VAR
IF (THIS^.isValueSpecial(currentValue)) THEN
	THIS^.assertionWasWrong(message, THIS^.getDebugInfo('valueIsNotSpecial'));
END_IF
END_METHOD

(*

short summary
=================
This assertion method checks if the current value is positve

.. attention::
	Any comparsion to NaN is ``FALSE`` that means if ``currentValue``
	is NaN then is the assertion false.
	For details check `IEEE 754`_.

.. attention::
	``currentValue`` has the value infinity means the assertion is true.
	``currentValue`` has the value -infinity means the assertion is false.
	``currentValue`` has the +0.0 means the assertion is true.
	``currentValue`` has the value -0.0 means the assertion is false.	
	For details check `IEEE 754`_.

.. _IEEE 754: https://en.wikipedia.org/wiki/IEEE_754

.. <legal notes>

legal notes
=================
| SPDX-FileCopyrightText: © 2022 ekvip automation GmbH <info@ekvip.de>
| SPDX-License-Identifier: Apache-2.0
| For details check: Apache-2.0_

.. _Apache-2.0: https://www.apache.org/licenses/LICENSE-2.0

.. </legal notes>

parameters
=================

*)

METHOD valueIsPositive
VAR_INPUT
	(* current value to check *)
	currentValue	:REAL;
	(* message if the assertion is false *)
	message			:AssertMessage;
END_VAR
VAR
	(* just to cast ``currentValue`` *)
	currentValueAsDWord	:POINTER TO DWORD;
END_VAR
IF (THIS^.isValueNaN(currentValue)) THEN	
	THIS^.assertionWasWrong(message, THIS^.getDebugInfo('valueIsPositive'));
ELSE
	currentValueAsDWord := ADR(currentValue);
	IF ((currentValueAsDWord^ AND THIS^.MASK_FOR_SIGN_BIT) = THIS^.MASK_FOR_SIGN_BIT) THEN
		THIS^.assertionWasWrong(message, THIS^.getDebugInfo('valueIsPositive'));
	END_IF
END_IF
END_METHOD

(*

short summary
=================
This assertion method checks if the current value is positive infinite
(infinty), for details check `IEEE 754`_

.. _IEEE 754: https://en.wikipedia.org/wiki/IEEE_754

.. <legal notes>

legal notes
=================
| SPDX-FileCopyrightText: © 2023 ekvip automation GmbH <info@ekvip.de>
| SPDX-License-Identifier: Apache-2.0
| For details check: Apache-2.0_

.. _Apache-2.0: https://www.apache.org/licenses/LICENSE-2.0

.. </legal notes>

parameters
=================

*)

METHOD valueIsPositiveInfinite
VAR_INPUT
	(* current value to check *)
	currentValue	:REAL;
	(* message if the assertion is false *)
	message			:AssertMessage;
END_VAR
IF (NOT THIS^.isValuePositiveInfinite(currentValue)) THEN
	THIS^.assertionWasWrong(message, THIS^.getDebugInfo('valueIsPositiveInfinite'));
END_IF
END_METHOD

(*

short summary
=================
This assertion method checks if the current value is -0.0
for details check `IEEE 754`_

.. _IEEE 754: https://en.wikipedia.org/wiki/IEEE_754

.. <legal notes>

legal notes
=================
| SPDX-FileCopyrightText: © 2023 ekvip automation GmbH <info@ekvip.de>
| SPDX-License-Identifier: Apache-2.0
| For details check: Apache-2.0_

.. _Apache-2.0: https://www.apache.org/licenses/LICENSE-2.0

.. </legal notes>

parameters
=================

*)

METHOD valueIsPositiveZero
VAR_INPUT
	(* current value to check *)
	currentValue	:REAL;
	(* message if the assertion is false *)
	message			:AssertMessage;
END_VAR
VAR
	(* just to cast ``currentValue`` *)
	currentValueAsDWord	:POINTER TO DWORD;
END_VAR
currentValueAsDWord := ADR(currentValue);
IF (currentValueAsDWord^ <> THIS^.ZERO) THEN
	THIS^.assertionWasWrong(message, THIS^.getDebugInfo('valueIsPositiveZero'));
END_IF
END_METHOD

(*

short summary
=================
This assertion method checks if the current value is a special
(NaN OR infinty OR -inifinity), for details check `IEEE 754`_

.. _IEEE 754: https://en.wikipedia.org/wiki/IEEE_754

.. <legal notes>

legal notes
=================
| SPDX-FileCopyrightText: © 2023 ekvip automation GmbH <info@ekvip.de>
| SPDX-License-Identifier: Apache-2.0
| For details check: Apache-2.0_

.. _Apache-2.0: https://www.apache.org/licenses/LICENSE-2.0

.. </legal notes>

parameters
=================

*)

METHOD valueIsSpecial
VAR_INPUT
	(* current value to check *)
	currentValue	:REAL;
	(* message if the assertion is false *)
	message			:AssertMessage;
END_VAR
IF (NOT THIS^.isValueSpecial(currentValue)) THEN
	THIS^.assertionWasWrong(message, THIS^.getDebugInfo('valueIsSpecial'));
END_IF
END_METHOD

(*

short summary
=================
This assertion method checks if the current value is a subnormal number
for details check `IEEE 754`_

.. _IEEE 754: https://en.wikipedia.org/wiki/IEEE_754

.. <legal notes>

legal notes
=================
| SPDX-FileCopyrightText: © 2023 ekvip automation GmbH <info@ekvip.de>
| SPDX-License-Identifier: Apache-2.0
| For details check: Apache-2.0_

.. _Apache-2.0: https://www.apache.org/licenses/LICENSE-2.0

.. </legal notes>

parameters
=================

*)

METHOD valueIsSubnormal
VAR_INPUT
	(* current value to check *)
	currentValue	:REAL;
	(* message if the assertion is false *)
	message			:AssertMessage;
END_VAR
VAR
	(* just to cast ``currentValue`` *)
	currentValueAsDWord	:POINTER TO DWORD;
END_VAR
IF (THIS^.isValueNaN(currentValue)) THEN
	THIS^.assertionWasWrong(message, THIS^.getDebugInfo('valueIsSubnormal'));
ELSE
	currentValueAsDWord := ADR(currentValue);
	IF ((currentValueAsDWord^ AND THIS^.MASK_FOR_EXPONENT) <> THIS^.ZERO) THEN
		THIS^.assertionWasWrong(message, THIS^.getDebugInfo('valueIsSubnormal'));
	END_IF
END_IF
END_METHOD

END_FUNCTION_BLOCK

// ---- Assertor/Assertions/FloatAssertions/Lreal/classes/LrealAssertions.TcPOU
(*

short summary
=================
This class provides assert statements for 64 bit floatings (``LREAL``).
It implements the interface :ref:`ILRealAssertions`

.. <legal notes>

legal notes
=================
| SPDX-FileCopyrightText: © 2022 ekvip automation GmbH <info@ekvip.de>
| SPDX-License-Identifier: Apache-2.0
| For details check: Apache-2.0_

.. _Apache-2.0: https://www.apache.org/licenses/LICENSE-2.0

.. </legal notes>

methods and properties
=======================

*)

{attribute 'reflection'}
FUNCTION_BLOCK INTERNAL LrealAssertions EXTENDS AbstactAssertion IMPLEMENTS ILRealAssertions
VAR
END_VAR
VAR CONSTANT
	(* mask for determining value as a special value *)
	MASK_FOR_EXPONENT 	:LWORD := 16#7FF0_0000_0000_0000;
	(* mask for determining a special value as NaN or infinite *)  
	MASK_FOR_FRACTION	:LWORD := 16#000F_FFFF_FFFF_FFFF;
	(* mask to get the sign bit of an infinite or zero value *)
	MASK_FOR_SIGN_BIT	:LWORD := 16#8000_0000_0000_0000;
	(* just to compare results or the memory of a float value *)
	ZERO				:DWORD := 16#0000_0000_0000_0000;
END_VAR

(*

short summary
=================
This abstract property returns the class name of the concrete object, 
It's for debugging purpose

.. <legal notes>

legal notes
=================
| SPDX-FileCopyrightText: © 2022 ekvip automation GmbH <info@ekvip.de>
| SPDX-License-Identifier: Apache-2.0
| For details check: Apache-2.0_

.. _Apache-2.0: https://www.apache.org/licenses/LICENSE-2.0

.. </legal notes>

*)

PROPERTY className :CNM_AbstractObject.ClassName
GET
className := 'CNM_AssertionInterfaceLib.LrealAssertions';
END_GET
END_PROPERTY

(*

short summary
=================
This method checks if a value is infinite
(infinty OR -inifinity), for details check `IEEE 754`_

.. _IEEE 754: https://en.wikipedia.org/wiki/IEEE_754

.. <legal notes>

legal notes
=================
| SPDX-FileCopyrightText: © 2023 ekvip automation GmbH <info@ekvip.de>
| SPDX-License-Identifier: Apache-2.0
| For details check: Apache-2.0_

.. _Apache-2.0: https://www.apache.org/licenses/LICENSE-2.0

.. </legal notes>

parameters
=================
:return: 
``TRUE``: value is inifinty or -infinity
``FALSE``: value is not inifinty and not -infinity

*)

METHOD PROTECTED isValueInfinite :BOOL
VAR_INPUT
	(* value to check *)
	value			:LREAL;	
END_VAR
VAR
	(* just to cast the value*)
	lrealAsLword	:POINTER TO LWORD;
END_VAR
lrealAsLword := ADR(value);
isValueInfinite := (
	THIS^.isValueSpecial(value)
	AND ((lrealAsLword^ AND THIS^.MASK_FOR_FRACTION) = THIS^.ZERO)
);
END_METHOD

(*

short summary
=================
This method checks if a value is not a number
(NaN), for details check `IEEE 754`_

.. _IEEE 754: https://en.wikipedia.org/wiki/IEEE_754

.. <legal notes>

legal notes
=================
| SPDX-FileCopyrightText: © 2023 ekvip automation GmbH <info@ekvip.de>
| SPDX-License-Identifier: Apache-2.0
| For details check: Apache-2.0_

.. _Apache-2.0: https://www.apache.org/licenses/LICENSE-2.0

.. </legal notes>

parameters
=================
:return: 
``TRUE``: value is NaN
``FALSE``: value is not NaN

*)

